  gc_DbmTranslation_de_Texts : ARRAY[0..2371] OF POINTER TO WSTRING(123) := [ADR(gc_DbmTranslation_de_Text0), ADR(gc_DbmTranslation_de_Text1), ADR(gc_DbmTranslation_de_Text2), ADR(gc_DbmTranslation_de_Text3), ADR(gc_DbmTranslation_de_Text4), ADR(gc_DbmTranslation_de_Text5), ADR(gc_DbmTranslation_de_Text6), ADR(gc_DbmTranslation_de_Text7), ADR(gc_DbmTranslation_de_Text8), ADR(gc_DbmTranslation_de_Text9), ADR(gc_DbmTranslation_de_Text10), ADR(gc_DbmTranslation_de_Text11), ADR(gc_DbmTranslation_de_Text12), ADR(gc_DbmTranslation_de_Text13), ADR(gc_DbmTranslation_de_Text14), ADR(gc_DbmTranslation_de_Text15), ADR(gc_DbmTranslation_de_Text16), ADR(gc_DbmTranslation_de_Text17), ADR(gc_DbmTranslation_de_Text18), ADR(gc_DbmTranslation_de_Text19), ADR(gc_DbmTranslation_de_Text20), ADR(gc_DbmTranslation_de_Text21), ADR(gc_DbmTranslation_de_Text22), ADR(gc_DbmTranslation_de_Text23), ADR(gc_DbmTranslation_de_Text24), ADR(gc_DbmTranslation_de_Text25), ADR(gc_DbmTranslation_de_Text26), ADR(gc_DbmTranslation_de_Text27), ADR(gc_DbmTranslation_de_Text28), ADR(gc_DbmTranslation_de_Text29), ADR(gc_DbmTranslation_de_Text30), ADR(gc_DbmTranslation_de_Text31), ADR(gc_DbmTranslation_de_Text32), ADR(gc_DbmTranslation_de_Text33), ADR(gc_DbmTranslation_de_Text34), ADR(gc_DbmTranslation_de_Text35), ADR(gc_DbmTranslation_de_Text36), ADR(gc_DbmTranslation_de_Text37), ADR(gc_DbmTranslation_de_Text38), ADR(gc_DbmTranslation_de_Text39), ADR(gc_DbmTranslation_de_Text40), ADR(gc_DbmTranslation_de_Text41), ADR(gc_DbmTranslation_de_Text42), ADR(gc_DbmTranslation_de_Text43), ADR(gc_DbmTranslation_de_Text44), ADR(gc_DbmTranslation_de_Text45), ADR(gc_DbmTranslation_de_Text46), ADR(gc_DbmTranslation_de_Text47), ADR(gc_DbmTranslation_de_Text48), ADR(gc_DbmTranslation_de_Text49), ADR(gc_DbmTranslation_de_Text50), ADR(gc_DbmTranslation_de_Text51), ADR(gc_DbmTranslation_de_Text52), ADR(gc_DbmTranslation_de_Text53), ADR(gc_DbmTranslation_de_Text54), ADR(gc_DbmTranslation_de_Text55), ADR(gc_DbmTranslation_de_Text56), ADR(gc_DbmTranslation_de_Text57), ADR(gc_DbmTranslation_de_Text58), ADR(gc_DbmTranslation_de_Text59), ADR(gc_DbmTranslation_de_Text60), ADR(gc_DbmTranslation_de_Text61), ADR(gc_DbmTranslation_de_Text62), ADR(gc_DbmTranslation_de_Text63), ADR(gc_DbmTranslation_de_Text64), ADR(gc_DbmTranslation_de_Text65), ADR(gc_DbmTranslation_de_Text66), ADR(gc_DbmTranslation_de_Text67), ADR(gc_DbmTranslation_de_Text68), ADR(gc_DbmTranslation_de_Text69), ADR(gc_DbmTranslation_de_Text70), ADR(gc_DbmTranslation_de_Text71), ADR(gc_DbmTranslation_de_Text72), ADR(gc_DbmTranslation_de_Text73), ADR(gc_DbmTranslation_de_Text74), ADR(gc_DbmTranslation_de_Text75), ADR(gc_DbmTranslation_de_Text76), ADR(gc_DbmTranslation_de_Text77), ADR(gc_DbmTranslation_de_Text78), ADR(gc_DbmTranslation_de_Text79), ADR(gc_DbmTranslation_de_Text80), ADR(gc_DbmTranslation_de_Text81), ADR(gc_DbmTranslation_de_Text82), ADR(gc_DbmTranslation_de_Text83), ADR(gc_DbmTranslation_de_Text84), ADR(gc_DbmTranslation_de_Text85), ADR(gc_DbmTranslation_de_Text86), ADR(gc_DbmTranslation_de_Text87), ADR(gc_DbmTranslation_de_Text88), ADR(gc_DbmTranslation_de_Text89), ADR(gc_DbmTranslation_de_Text90), ADR(gc_DbmTranslation_de_Text91), ADR(gc_DbmTranslation_de_Text92), ADR(gc_DbmTranslation_de_Text93), ADR(gc_DbmTranslation_de_Text94), ADR(gc_DbmTranslation_de_Text95), ADR(gc_DbmTranslation_de_Text96), ADR(gc_DbmTranslation_de_Text97), ADR(gc_DbmTranslation_de_Text98), ADR(gc_DbmTranslation_de_Text99), ADR(gc_DbmTranslation_de_Text100), ADR(gc_DbmTranslation_de_Text101), ADR(gc_DbmTranslation_de_Text102), ADR(gc_DbmTranslation_de_Text103), ADR(gc_DbmTranslation_de_Text104), ADR(gc_DbmTranslation_de_Text105), ADR(gc_DbmTranslation_de_Text106), ADR(gc_DbmTranslation_de_Text107), ADR(gc_DbmTranslation_de_Text108), ADR(gc_DbmTranslation_de_Text109), ADR(gc_DbmTranslation_de_Text110), ADR(gc_DbmTranslation_de_Text111), ADR(gc_DbmTranslation_de_Text112), ADR(gc_DbmTranslation_de_Text113), ADR(gc_DbmTranslation_de_Text114), ADR(gc_DbmTranslation_de_Text115), ADR(gc_DbmTranslation_de_Text116), ADR(gc_DbmTranslation_de_Text117), ADR(gc_DbmTranslation_de_Text118), ADR(gc_DbmTranslation_de_Text119), ADR(gc_DbmTranslation_de_Text120), ADR(gc_DbmTranslation_de_Text121), ADR(gc_DbmTranslation_de_Text122), ADR(gc_DbmTranslation_de_Text123), ADR(gc_DbmTranslation_de_Text124), ADR(gc_DbmTranslation_de_Text125), ADR(gc_DbmTranslation_de_Text126), ADR(gc_DbmTranslation_de_Text127), ADR(gc_DbmTranslation_de_Text128), ADR(gc_DbmTranslation_de_Text129), ADR(gc_DbmTranslation_de_Text130), ADR(gc_DbmTranslation_de_Text131), ADR(gc_DbmTranslation_de_Text132), ADR(gc_DbmTranslation_de_Text133), ADR(gc_DbmTranslation_de_Text134), ADR(gc_DbmTranslation_de_Text135), ADR(gc_DbmTranslation_de_Text136), ADR(gc_DbmTranslation_de_Text137), ADR(gc_DbmTranslation_de_Text138), ADR(gc_DbmTranslation_de_Text139), ADR(gc_DbmTranslation_de_Text140), ADR(gc_DbmTranslation_de_Text141), ADR(gc_DbmTranslation_de_Text142), ADR(gc_DbmTranslation_de_Text143), ADR(gc_DbmTranslation_de_Text144), ADR(gc_DbmTranslation_de_Text145), ADR(gc_DbmTranslation_de_Text146), ADR(gc_DbmTranslation_de_Text147), ADR(gc_DbmTranslation_de_Text148), ADR(gc_DbmTranslation_de_Text149), ADR(gc_DbmTranslation_de_Text150), ADR(gc_DbmTranslation_de_Text151), ADR(gc_DbmTranslation_de_Text152), ADR(gc_DbmTranslation_de_Text153), ADR(gc_DbmTranslation_de_Text154), ADR(gc_DbmTranslation_de_Text155), ADR(gc_DbmTranslation_de_Text156), ADR(gc_DbmTranslation_de_Text157), ADR(gc_DbmTranslation_de_Text158), ADR(gc_DbmTranslation_de_Text159), ADR(gc_DbmTranslation_de_Text160), ADR(gc_DbmTranslation_de_Text161), ADR(gc_DbmTranslation_de_Text162), ADR(gc_DbmTranslation_de_Text163), ADR(gc_DbmTranslation_de_Text164), ADR(gc_DbmTranslation_de_Text165), ADR(gc_DbmTranslation_de_Text166), ADR(gc_DbmTranslation_de_Text167), ADR(gc_DbmTranslation_de_Text168), ADR(gc_DbmTranslation_de_Text169), ADR(gc_DbmTranslation_de_Text170), ADR(gc_DbmTranslation_de_Text171), ADR(gc_DbmTranslation_de_Text172), ADR(gc_DbmTranslation_de_Text173), ADR(gc_DbmTranslation_de_Text174), ADR(gc_DbmTranslation_de_Text175), ADR(gc_DbmTranslation_de_Text176), ADR(gc_DbmTranslation_de_Text177), ADR(gc_DbmTranslation_de_Text178), ADR(gc_DbmTranslation_de_Text179), ADR(gc_DbmTranslation_de_Text180), ADR(gc_DbmTranslation_de_Text181), ADR(gc_DbmTranslation_de_Text182), ADR(gc_DbmTranslation_de_Text183), ADR(gc_DbmTranslation_de_Text184), ADR(gc_DbmTranslation_de_Text185), ADR(gc_DbmTranslation_de_Text186), ADR(gc_DbmTranslation_de_Text187), ADR(gc_DbmTranslation_de_Text188), ADR(gc_DbmTranslation_de_Text189), ADR(gc_DbmTranslation_de_Text190), ADR(gc_DbmTranslation_de_Text191), ADR(gc_DbmTranslation_de_Text192), ADR(gc_DbmTranslation_de_Text193), ADR(gc_DbmTranslation_de_Text194), ADR(gc_DbmTranslation_de_Text195), ADR(gc_DbmTranslation_de_Text196), ADR(gc_DbmTranslation_de_Text197), ADR(gc_DbmTranslation_de_Text198), ADR(gc_DbmTranslation_de_Text199), ADR(gc_DbmTranslation_de_Text200), ADR(gc_DbmTranslation_de_Text201), ADR(gc_DbmTranslation_de_Text202), ADR(gc_DbmTranslation_de_Text203), ADR(gc_DbmTranslation_de_Text204), ADR(gc_DbmTranslation_de_Text205), ADR(gc_DbmTranslation_de_Text206), ADR(gc_DbmTranslation_de_Text207), ADR(gc_DbmTranslation_de_Text208), ADR(gc_DbmTranslation_de_Text209), ADR(gc_DbmTranslation_de_Text210), ADR(gc_DbmTranslation_de_Text211), ADR(gc_DbmTranslation_de_Text212), ADR(gc_DbmTranslation_de_Text213), ADR(gc_DbmTranslation_de_Text214), ADR(gc_DbmTranslation_de_Text215), ADR(gc_DbmTranslation_de_Text216), ADR(gc_DbmTranslation_de_Text217), ADR(gc_DbmTranslation_de_Text218), ADR(gc_DbmTranslation_de_Text219), ADR(gc_DbmTranslation_de_Text220), ADR(gc_DbmTranslation_de_Text221), ADR(gc_DbmTranslation_de_Text222), ADR(gc_DbmTranslation_de_Text223), ADR(gc_DbmTranslation_de_Text224), ADR(gc_DbmTranslation_de_Text225), ADR(gc_DbmTranslation_de_Text226), ADR(gc_DbmTranslation_de_Text227), ADR(gc_DbmTranslation_de_Text228), ADR(gc_DbmTranslation_de_Text229), ADR(gc_DbmTranslation_de_Text230), ADR(gc_DbmTranslation_de_Text231), ADR(gc_DbmTranslation_de_Text232), ADR(gc_DbmTranslation_de_Text233), ADR(gc_DbmTranslation_de_Text234), ADR(gc_DbmTranslation_de_Text235), ADR(gc_DbmTranslation_de_Text236), ADR(gc_DbmTranslation_de_Text237), ADR(gc_DbmTranslation_de_Text238), ADR(gc_DbmTranslation_de_Text239), ADR(gc_DbmTranslation_de_Text240), ADR(gc_DbmTranslation_de_Text241), ADR(gc_DbmTranslation_de_Text242), ADR(gc_DbmTranslation_de_Text243), ADR(gc_DbmTranslation_de_Text244), ADR(gc_DbmTranslation_de_Text245), ADR(gc_DbmTranslation_de_Text246), ADR(gc_DbmTranslation_de_Text247), ADR(gc_DbmTranslation_de_Text248), ADR(gc_DbmTranslation_de_Text249), ADR(gc_DbmTranslation_de_Text250), ADR(gc_DbmTranslation_de_Text251), ADR(gc_DbmTranslation_de_Text252), ADR(gc_DbmTranslation_de_Text253), ADR(gc_DbmTranslation_de_Text254), ADR(gc_DbmTranslation_de_Text255), ADR(gc_DbmTranslation_de_Text256), ADR(gc_DbmTranslation_de_Text257), ADR(gc_DbmTranslation_de_Text258), ADR(gc_DbmTranslation_de_Text259), ADR(gc_DbmTranslation_de_Text260), ADR(gc_DbmTranslation_de_Text261), ADR(gc_DbmTranslation_de_Text262), ADR(gc_DbmTranslation_de_Text263), ADR(gc_DbmTranslation_de_Text264), ADR(gc_DbmTranslation_de_Text265), ADR(gc_DbmTranslation_de_Text266), ADR(gc_DbmTranslation_de_Text267), ADR(gc_DbmTranslation_de_Text268), ADR(gc_DbmTranslation_de_Text269), ADR(gc_DbmTranslation_de_Text270), ADR(gc_DbmTranslation_de_Text271), ADR(gc_DbmTranslation_de_Text272), ADR(gc_DbmTranslation_de_Text273), ADR(gc_DbmTranslation_de_Text274), ADR(gc_DbmTranslation_de_Text275), ADR(gc_DbmTranslation_de_Text276), ADR(gc_DbmTranslation_de_Text277), ADR(gc_DbmTranslation_de_Text278), ADR(gc_DbmTranslation_de_Text279), ADR(gc_DbmTranslation_de_Text280), ADR(gc_DbmTranslation_de_Text281), ADR(gc_DbmTranslation_de_Text282), ADR(gc_DbmTranslation_de_Text283), ADR(gc_DbmTranslation_de_Text284), ADR(gc_DbmTranslation_de_Text285), ADR(gc_DbmTranslation_de_Text286), ADR(gc_DbmTranslation_de_Text287), ADR(gc_DbmTranslation_de_Text288), ADR(gc_DbmTranslation_de_Text289), ADR(gc_DbmTranslation_de_Text290), ADR(gc_DbmTranslation_de_Text291), ADR(gc_DbmTranslation_de_Text292), ADR(gc_DbmTranslation_de_Text293), ADR(gc_DbmTranslation_de_Text294), ADR(gc_DbmTranslation_de_Text295), ADR(gc_DbmTranslation_de_Text296), ADR(gc_DbmTranslation_de_Text297), ADR(gc_DbmTranslation_de_Text298), ADR(gc_DbmTranslation_de_Text299), ADR(gc_DbmTranslation_de_Text300), ADR(gc_DbmTranslation_de_Text301), ADR(gc_DbmTranslation_de_Text302), ADR(gc_DbmTranslation_de_Text303), ADR(gc_DbmTranslation_de_Text304), ADR(gc_DbmTranslation_de_Text305), ADR(gc_DbmTranslation_de_Text306), ADR(gc_DbmTranslation_de_Text307), ADR(gc_DbmTranslation_de_Text308), ADR(gc_DbmTranslation_de_Text309), ADR(gc_DbmTranslation_de_Text310), ADR(gc_DbmTranslation_de_Text311), ADR(gc_DbmTranslation_de_Text312), ADR(gc_DbmTranslation_de_Text313), ADR(gc_DbmTranslation_de_Text314), ADR(gc_DbmTranslation_de_Text315), ADR(gc_DbmTranslation_de_Text316), ADR(gc_DbmTranslation_de_Text317), ADR(gc_DbmTranslation_de_Text318), ADR(gc_DbmTranslation_de_Text319), ADR(gc_DbmTranslation_de_Text320), ADR(gc_DbmTranslation_de_Text321), ADR(gc_DbmTranslation_de_Text322), ADR(gc_DbmTranslation_de_Text323), ADR(gc_DbmTranslation_de_Text324), ADR(gc_DbmTranslation_de_Text325), ADR(gc_DbmTranslation_de_Text326), ADR(gc_DbmTranslation_de_Text327), ADR(gc_DbmTranslation_de_Text328), ADR(gc_DbmTranslation_de_Text329), ADR(gc_DbmTranslation_de_Text330), ADR(gc_DbmTranslation_de_Text331), ADR(gc_DbmTranslation_de_Text332), ADR(gc_DbmTranslation_de_Text333), ADR(gc_DbmTranslation_de_Text334), ADR(gc_DbmTranslation_de_Text335), ADR(gc_DbmTranslation_de_Text336), ADR(gc_DbmTranslation_de_Text337), ADR(gc_DbmTranslation_de_Text338), ADR(gc_DbmTranslation_de_Text339), ADR(gc_DbmTranslation_de_Text340), ADR(gc_DbmTranslation_de_Text341), ADR(gc_DbmTranslation_de_Text342), ADR(gc_DbmTranslation_de_Text343), ADR(gc_DbmTranslation_de_Text344), ADR(gc_DbmTranslation_de_Text345), ADR(gc_DbmTranslation_de_Text346), ADR(gc_DbmTranslation_de_Text347), ADR(gc_DbmTranslation_de_Text348), ADR(gc_DbmTranslation_de_Text349), ADR(gc_DbmTranslation_de_Text350), ADR(gc_DbmTranslation_de_Text351), ADR(gc_DbmTranslation_de_Text352), ADR(gc_DbmTranslation_de_Text353), ADR(gc_DbmTranslation_de_Text354), ADR(gc_DbmTranslation_de_Text355), ADR(gc_DbmTranslation_de_Text356), ADR(gc_DbmTranslation_de_Text357), ADR(gc_DbmTranslation_de_Text358), ADR(gc_DbmTranslation_de_Text359), ADR(gc_DbmTranslation_de_Text360), ADR(gc_DbmTranslation_de_Text361), ADR(gc_DbmTranslation_de_Text362), ADR(gc_DbmTranslation_de_Text363), ADR(gc_DbmTranslation_de_Text364), ADR(gc_DbmTranslation_de_Text365), ADR(gc_DbmTranslation_de_Text366), ADR(gc_DbmTranslation_de_Text367), ADR(gc_DbmTranslation_de_Text368), ADR(gc_DbmTranslation_de_Text369), ADR(gc_DbmTranslation_de_Text370), ADR(gc_DbmTranslation_de_Text371), ADR(gc_DbmTranslation_de_Text372), ADR(gc_DbmTranslation_de_Text373), ADR(gc_DbmTranslation_de_Text374), ADR(gc_DbmTranslation_de_Text375), ADR(gc_DbmTranslation_de_Text376), ADR(gc_DbmTranslation_de_Text377), ADR(gc_DbmTranslation_de_Text378), ADR(gc_DbmTranslation_de_Text379), ADR(gc_DbmTranslation_de_Text380), ADR(gc_DbmTranslation_de_Text381), ADR(gc_DbmTranslation_de_Text382), ADR(gc_DbmTranslation_de_Text383), ADR(gc_DbmTranslation_de_Text384), ADR(gc_DbmTranslation_de_Text385), ADR(gc_DbmTranslation_de_Text386), ADR(gc_DbmTranslation_de_Text387), ADR(gc_DbmTranslation_de_Text388), ADR(gc_DbmTranslation_de_Text389), ADR(gc_DbmTranslation_de_Text390), ADR(gc_DbmTranslation_de_Text391), ADR(gc_DbmTranslation_de_Text392), ADR(gc_DbmTranslation_de_Text393), ADR(gc_DbmTranslation_de_Text394), ADR(gc_DbmTranslation_de_Text395), ADR(gc_DbmTranslation_de_Text396), ADR(gc_DbmTranslation_de_Text397), ADR(gc_DbmTranslation_de_Text398), ADR(gc_DbmTranslation_de_Text399), ADR(gc_DbmTranslation_de_Text400), ADR(gc_DbmTranslation_de_Text401), ADR(gc_DbmTranslation_de_Text402), ADR(gc_DbmTranslation_de_Text403), ADR(gc_DbmTranslation_de_Text404), ADR(gc_DbmTranslation_de_Text405), ADR(gc_DbmTranslation_de_Text406), ADR(gc_DbmTranslation_de_Text407), ADR(gc_DbmTranslation_de_Text408), ADR(gc_DbmTranslation_de_Text409), ADR(gc_DbmTranslation_de_Text410), ADR(gc_DbmTranslation_de_Text411), ADR(gc_DbmTranslation_de_Text412), ADR(gc_DbmTranslation_de_Text413), ADR(gc_DbmTranslation_de_Text414), ADR(gc_DbmTranslation_de_Text415), ADR(gc_DbmTranslation_de_Text416), ADR(gc_DbmTranslation_de_Text417), ADR(gc_DbmTranslation_de_Text418), ADR(gc_DbmTranslation_de_Text419), ADR(gc_DbmTranslation_de_Text420), ADR(gc_DbmTranslation_de_Text421), ADR(gc_DbmTranslation_de_Text422), ADR(gc_DbmTranslation_de_Text423), ADR(gc_DbmTranslation_de_Text424), ADR(gc_DbmTranslation_de_Text425), ADR(gc_DbmTranslation_de_Text426), ADR(gc_DbmTranslation_de_Text427), ADR(gc_DbmTranslation_de_Text428), ADR(gc_DbmTranslation_de_Text429), ADR(gc_DbmTranslation_de_Text430), ADR(gc_DbmTranslation_de_Text431), ADR(gc_DbmTranslation_de_Text432), ADR(gc_DbmTranslation_de_Text433), ADR(gc_DbmTranslation_de_Text434), ADR(gc_DbmTranslation_de_Text435), ADR(gc_DbmTranslation_de_Text436), ADR(gc_DbmTranslation_de_Text437), ADR(gc_DbmTranslation_de_Text438), ADR(gc_DbmTranslation_de_Text439), ADR(gc_DbmTranslation_de_Text440), ADR(gc_DbmTranslation_de_Text441), ADR(gc_DbmTranslation_de_Text442), ADR(gc_DbmTranslation_de_Text443), ADR(gc_DbmTranslation_de_Text444), ADR(gc_DbmTranslation_de_Text445), ADR(gc_DbmTranslation_de_Text446), ADR(gc_DbmTranslation_de_Text447), ADR(gc_DbmTranslation_de_Text448), ADR(gc_DbmTranslation_de_Text449), ADR(gc_DbmTranslation_de_Text450), ADR(gc_DbmTranslation_de_Text451), ADR(gc_DbmTranslation_de_Text452), ADR(gc_DbmTranslation_de_Text453), ADR(gc_DbmTranslation_de_Text454), ADR(gc_DbmTranslation_de_Text455), ADR(gc_DbmTranslation_de_Text456), ADR(gc_DbmTranslation_de_Text457), ADR(gc_DbmTranslation_de_Text458), ADR(gc_DbmTranslation_de_Text459), ADR(gc_DbmTranslation_de_Text460), ADR(gc_DbmTranslation_de_Text461), ADR(gc_DbmTranslation_de_Text462), ADR(gc_DbmTranslation_de_Text463), ADR(gc_DbmTranslation_de_Text464), ADR(gc_DbmTranslation_de_Text465), ADR(gc_DbmTranslation_de_Text466), ADR(gc_DbmTranslation_de_Text467), ADR(gc_DbmTranslation_de_Text468), ADR(gc_DbmTranslation_de_Text469), ADR(gc_DbmTranslation_de_Text470), ADR(gc_DbmTranslation_de_Text471), ADR(gc_DbmTranslation_de_Text472), ADR(gc_DbmTranslation_de_Text473), ADR(gc_DbmTranslation_de_Text474), ADR(gc_DbmTranslation_de_Text475), ADR(gc_DbmTranslation_de_Text476), ADR(gc_DbmTranslation_de_Text477), ADR(gc_DbmTranslation_de_Text478), ADR(gc_DbmTranslation_de_Text479), ADR(gc_DbmTranslation_de_Text480), ADR(gc_DbmTranslation_de_Text481), ADR(gc_DbmTranslation_de_Text482), ADR(gc_DbmTranslation_de_Text483), ADR(gc_DbmTranslation_de_Text484), ADR(gc_DbmTranslation_de_Text485), ADR(gc_DbmTranslation_de_Text486), ADR(gc_DbmTranslation_de_Text487), ADR(gc_DbmTranslation_de_Text488), ADR(gc_DbmTranslation_de_Text489), ADR(gc_DbmTranslation_de_Text490), ADR(gc_DbmTranslation_de_Text491), ADR(gc_DbmTranslation_de_Text492), ADR(gc_DbmTranslation_de_Text493), ADR(gc_DbmTranslation_de_Text494), ADR(gc_DbmTranslation_de_Text495), ADR(gc_DbmTranslation_de_Text496), ADR(gc_DbmTranslation_de_Text497), ADR(gc_DbmTranslation_de_Text498), ADR(gc_DbmTranslation_de_Text499), ADR(gc_DbmTranslation_de_Text500), ADR(gc_DbmTranslation_de_Text501), ADR(gc_DbmTranslation_de_Text502), ADR(gc_DbmTranslation_de_Text503), ADR(gc_DbmTranslation_de_Text504), ADR(gc_DbmTranslation_de_Text505), ADR(gc_DbmTranslation_de_Text506), ADR(gc_DbmTranslation_de_Text507), ADR(gc_DbmTranslation_de_Text508), ADR(gc_DbmTranslation_de_Text509), ADR(gc_DbmTranslation_de_Text510), ADR(gc_DbmTranslation_de_Text511), ADR(gc_DbmTranslation_de_Text512), ADR(gc_DbmTranslation_de_Text513), ADR(gc_DbmTranslation_de_Text514), ADR(gc_DbmTranslation_de_Text515), ADR(gc_DbmTranslation_de_Text516), ADR(gc_DbmTranslation_de_Text517), ADR(gc_DbmTranslation_de_Text518), ADR(gc_DbmTranslation_de_Text519), ADR(gc_DbmTranslation_de_Text520), ADR(gc_DbmTranslation_de_Text521), ADR(gc_DbmTranslation_de_Text522), ADR(gc_DbmTranslation_de_Text523), ADR(gc_DbmTranslation_de_Text524), ADR(gc_DbmTranslation_de_Text525), ADR(gc_DbmTranslation_de_Text526), ADR(gc_DbmTranslation_de_Text527), ADR(gc_DbmTranslation_de_Text528), ADR(gc_DbmTranslation_de_Text529), ADR(gc_DbmTranslation_de_Text530), ADR(gc_DbmTranslation_de_Text531), ADR(gc_DbmTranslation_de_Text532), ADR(gc_DbmTranslation_de_Text533), ADR(gc_DbmTranslation_de_Text534), ADR(gc_DbmTranslation_de_Text535), ADR(gc_DbmTranslation_de_Text536), ADR(gc_DbmTranslation_de_Text537), ADR(gc_DbmTranslation_de_Text538), ADR(gc_DbmTranslation_de_Text539), ADR(gc_DbmTranslation_de_Text540), ADR(gc_DbmTranslation_de_Text541), ADR(gc_DbmTranslation_de_Text542), ADR(gc_DbmTranslation_de_Text543), ADR(gc_DbmTranslation_de_Text544), ADR(gc_DbmTranslation_de_Text545), ADR(gc_DbmTranslation_de_Text546), ADR(gc_DbmTranslation_de_Text547), ADR(gc_DbmTranslation_de_Text548), ADR(gc_DbmTranslation_de_Text549), ADR(gc_DbmTranslation_de_Text550), ADR(gc_DbmTranslation_de_Text551), ADR(gc_DbmTranslation_de_Text552), ADR(gc_DbmTranslation_de_Text553), ADR(gc_DbmTranslation_de_Text554), ADR(gc_DbmTranslation_de_Text555), ADR(gc_DbmTranslation_de_Text556), ADR(gc_DbmTranslation_de_Text557), ADR(gc_DbmTranslation_de_Text558), ADR(gc_DbmTranslation_de_Text559), ADR(gc_DbmTranslation_de_Text560), ADR(gc_DbmTranslation_de_Text561), ADR(gc_DbmTranslation_de_Text562), ADR(gc_DbmTranslation_de_Text563), ADR(gc_DbmTranslation_de_Text564), ADR(gc_DbmTranslation_de_Text565), ADR(gc_DbmTranslation_de_Text566), ADR(gc_DbmTranslation_de_Text567), ADR(gc_DbmTranslation_de_Text568), ADR(gc_DbmTranslation_de_Text569), ADR(gc_DbmTranslation_de_Text570), ADR(gc_DbmTranslation_de_Text571), ADR(gc_DbmTranslation_de_Text572), ADR(gc_DbmTranslation_de_Text573), ADR(gc_DbmTranslation_de_Text574), ADR(gc_DbmTranslation_de_Text575), ADR(gc_DbmTranslation_de_Text576), ADR(gc_DbmTranslation_de_Text577), ADR(gc_DbmTranslation_de_Text578), ADR(gc_DbmTranslation_de_Text579), ADR(gc_DbmTranslation_de_Text580), ADR(gc_DbmTranslation_de_Text581), ADR(gc_DbmTranslation_de_Text582), ADR(gc_DbmTranslation_de_Text583), ADR(gc_DbmTranslation_de_Text584), ADR(gc_DbmTranslation_de_Text585), ADR(gc_DbmTranslation_de_Text586), ADR(gc_DbmTranslation_de_Text587), ADR(gc_DbmTranslation_de_Text588), ADR(gc_DbmTranslation_de_Text589), ADR(gc_DbmTranslation_de_Text590), ADR(gc_DbmTranslation_de_Text591), ADR(gc_DbmTranslation_de_Text592), ADR(gc_DbmTranslation_de_Text593), ADR(gc_DbmTranslation_de_Text594), ADR(gc_DbmTranslation_de_Text595), ADR(gc_DbmTranslation_de_Text596), ADR(gc_DbmTranslation_de_Text597), ADR(gc_DbmTranslation_de_Text598), ADR(gc_DbmTranslation_de_Text599), ADR(gc_DbmTranslation_de_Text600), ADR(gc_DbmTranslation_de_Text601), ADR(gc_DbmTranslation_de_Text602), ADR(gc_DbmTranslation_de_Text603), ADR(gc_DbmTranslation_de_Text604), ADR(gc_DbmTranslation_de_Text605), ADR(gc_DbmTranslation_de_Text606), ADR(gc_DbmTranslation_de_Text607), ADR(gc_DbmTranslation_de_Text608), ADR(gc_DbmTranslation_de_Text609), ADR(gc_DbmTranslation_de_Text610), ADR(gc_DbmTranslation_de_Text611), ADR(gc_DbmTranslation_de_Text612), ADR(gc_DbmTranslation_de_Text613), ADR(gc_DbmTranslation_de_Text614), ADR(gc_DbmTranslation_de_Text615), ADR(gc_DbmTranslation_de_Text616), ADR(gc_DbmTranslation_de_Text617), ADR(gc_DbmTranslation_de_Text618), ADR(gc_DbmTranslation_de_Text619), ADR(gc_DbmTranslation_de_Text620), ADR(gc_DbmTranslation_de_Text621), ADR(gc_DbmTranslation_de_Text622), ADR(gc_DbmTranslation_de_Text623), ADR(gc_DbmTranslation_de_Text624), ADR(gc_DbmTranslation_de_Text625), ADR(gc_DbmTranslation_de_Text626), ADR(gc_DbmTranslation_de_Text627), ADR(gc_DbmTranslation_de_Text628), ADR(gc_DbmTranslation_de_Text629), ADR(gc_DbmTranslation_de_Text630), ADR(gc_DbmTranslation_de_Text631), ADR(gc_DbmTranslation_de_Text632), ADR(gc_DbmTranslation_de_Text633), ADR(gc_DbmTranslation_de_Text634), ADR(gc_DbmTranslation_de_Text635), ADR(gc_DbmTranslation_de_Text636), ADR(gc_DbmTranslation_de_Text637), ADR(gc_DbmTranslation_de_Text638), ADR(gc_DbmTranslation_de_Text639), ADR(gc_DbmTranslation_de_Text640), ADR(gc_DbmTranslation_de_Text641), ADR(gc_DbmTranslation_de_Text642), ADR(gc_DbmTranslation_de_Text643), ADR(gc_DbmTranslation_de_Text644), ADR(gc_DbmTranslation_de_Text645), ADR(gc_DbmTranslation_de_Text646), ADR(gc_DbmTranslation_de_Text647), ADR(gc_DbmTranslation_de_Text648), ADR(gc_DbmTranslation_de_Text649), ADR(gc_DbmTranslation_de_Text650), ADR(gc_DbmTranslation_de_Text651), ADR(gc_DbmTranslation_de_Text652), ADR(gc_DbmTranslation_de_Text653), ADR(gc_DbmTranslation_de_Text654), ADR(gc_DbmTranslation_de_Text655), ADR(gc_DbmTranslation_de_Text656), ADR(gc_DbmTranslation_de_Text657), ADR(gc_DbmTranslation_de_Text658), ADR(gc_DbmTranslation_de_Text659), ADR(gc_DbmTranslation_de_Text660), ADR(gc_DbmTranslation_de_Text661), ADR(gc_DbmTranslation_de_Text662), ADR(gc_DbmTranslation_de_Text663), ADR(gc_DbmTranslation_de_Text664), ADR(gc_DbmTranslation_de_Text665), ADR(gc_DbmTranslation_de_Text666), ADR(gc_DbmTranslation_de_Text667), ADR(gc_DbmTranslation_de_Text668), ADR(gc_DbmTranslation_de_Text669), ADR(gc_DbmTranslation_de_Text670), ADR(gc_DbmTranslation_de_Text671), ADR(gc_DbmTranslation_de_Text672), ADR(gc_DbmTranslation_de_Text673), ADR(gc_DbmTranslation_de_Text674), ADR(gc_DbmTranslation_de_Text675), ADR(gc_DbmTranslation_de_Text676), ADR(gc_DbmTranslation_de_Text677), ADR(gc_DbmTranslation_de_Text678), ADR(gc_DbmTranslation_de_Text679), ADR(gc_DbmTranslation_de_Text680), ADR(gc_DbmTranslation_de_Text681), ADR(gc_DbmTranslation_de_Text682), ADR(gc_DbmTranslation_de_Text683), ADR(gc_DbmTranslation_de_Text684), ADR(gc_DbmTranslation_de_Text685), ADR(gc_DbmTranslation_de_Text686), ADR(gc_DbmTranslation_de_Text687), ADR(gc_DbmTranslation_de_Text688), ADR(gc_DbmTranslation_de_Text689), ADR(gc_DbmTranslation_de_Text690), ADR(gc_DbmTranslation_de_Text691), ADR(gc_DbmTranslation_de_Text692), ADR(gc_DbmTranslation_de_Text693), ADR(gc_DbmTranslation_de_Text694), ADR(gc_DbmTranslation_de_Text695), ADR(gc_DbmTranslation_de_Text696), ADR(gc_DbmTranslation_de_Text697), ADR(gc_DbmTranslation_de_Text698), ADR(gc_DbmTranslation_de_Text699), ADR(gc_DbmTranslation_de_Text700), ADR(gc_DbmTranslation_de_Text701), ADR(gc_DbmTranslation_de_Text702), ADR(gc_DbmTranslation_de_Text703), ADR(gc_DbmTranslation_de_Text704), ADR(gc_DbmTranslation_de_Text705), ADR(gc_DbmTranslation_de_Text706), ADR(gc_DbmTranslation_de_Text707), ADR(gc_DbmTranslation_de_Text708), ADR(gc_DbmTranslation_de_Text709), ADR(gc_DbmTranslation_de_Text710), ADR(gc_DbmTranslation_de_Text711), ADR(gc_DbmTranslation_de_Text712), ADR(gc_DbmTranslation_de_Text713), ADR(gc_DbmTranslation_de_Text714), ADR(gc_DbmTranslation_de_Text715), ADR(gc_DbmTranslation_de_Text716), ADR(gc_DbmTranslation_de_Text717), ADR(gc_DbmTranslation_de_Text718), ADR(gc_DbmTranslation_de_Text719), ADR(gc_DbmTranslation_de_Text720), ADR(gc_DbmTranslation_de_Text721), ADR(gc_DbmTranslation_de_Text722), ADR(gc_DbmTranslation_de_Text723), ADR(gc_DbmTranslation_de_Text724), ADR(gc_DbmTranslation_de_Text725), ADR(gc_DbmTranslation_de_Text726), ADR(gc_DbmTranslation_de_Text727), ADR(gc_DbmTranslation_de_Text728), ADR(gc_DbmTranslation_de_Text729), ADR(gc_DbmTranslation_de_Text730), ADR(gc_DbmTranslation_de_Text731), ADR(gc_DbmTranslation_de_Text732), ADR(gc_DbmTranslation_de_Text733), ADR(gc_DbmTranslation_de_Text734), ADR(gc_DbmTranslation_de_Text735), ADR(gc_DbmTranslation_de_Text736), ADR(gc_DbmTranslation_de_Text737), ADR(gc_DbmTranslation_de_Text738), ADR(gc_DbmTranslation_de_Text739), ADR(gc_DbmTranslation_de_Text740), ADR(gc_DbmTranslation_de_Text741), ADR(gc_DbmTranslation_de_Text742), ADR(gc_DbmTranslation_de_Text743), ADR(gc_DbmTranslation_de_Text744), ADR(gc_DbmTranslation_de_Text745), ADR(gc_DbmTranslation_de_Text746), ADR(gc_DbmTranslation_de_Text747), ADR(gc_DbmTranslation_de_Text748), ADR(gc_DbmTranslation_de_Text749), ADR(gc_DbmTranslation_de_Text750), ADR(gc_DbmTranslation_de_Text751), ADR(gc_DbmTranslation_de_Text752), ADR(gc_DbmTranslation_de_Text753), ADR(gc_DbmTranslation_de_Text754), ADR(gc_DbmTranslation_de_Text755), ADR(gc_DbmTranslation_de_Text756), ADR(gc_DbmTranslation_de_Text757), ADR(gc_DbmTranslation_de_Text758), ADR(gc_DbmTranslation_de_Text759), ADR(gc_DbmTranslation_de_Text760), ADR(gc_DbmTranslation_de_Text761), ADR(gc_DbmTranslation_de_Text762), ADR(gc_DbmTranslation_de_Text763), ADR(gc_DbmTranslation_de_Text764), ADR(gc_DbmTranslation_de_Text765), ADR(gc_DbmTranslation_de_Text766), ADR(gc_DbmTranslation_de_Text767), ADR(gc_DbmTranslation_de_Text768), ADR(gc_DbmTranslation_de_Text769), ADR(gc_DbmTranslation_de_Text770), ADR(gc_DbmTranslation_de_Text771), ADR(gc_DbmTranslation_de_Text772), ADR(gc_DbmTranslation_de_Text773), ADR(gc_DbmTranslation_de_Text774), ADR(gc_DbmTranslation_de_Text775), ADR(gc_DbmTranslation_de_Text776), ADR(gc_DbmTranslation_de_Text777), ADR(gc_DbmTranslation_de_Text778), ADR(gc_DbmTranslation_de_Text779), ADR(gc_DbmTranslation_de_Text780), ADR(gc_DbmTranslation_de_Text781), ADR(gc_DbmTranslation_de_Text782), ADR(gc_DbmTranslation_de_Text783), ADR(gc_DbmTranslation_de_Text784), ADR(gc_DbmTranslation_de_Text785), ADR(gc_DbmTranslation_de_Text786), ADR(gc_DbmTranslation_de_Text787), ADR(gc_DbmTranslation_de_Text788), ADR(gc_DbmTranslation_de_Text789), ADR(gc_DbmTranslation_de_Text790), ADR(gc_DbmTranslation_de_Text791), ADR(gc_DbmTranslation_de_Text792), ADR(gc_DbmTranslation_de_Text793), ADR(gc_DbmTranslation_de_Text794), ADR(gc_DbmTranslation_de_Text795), ADR(gc_DbmTranslation_de_Text796), ADR(gc_DbmTranslation_de_Text797), ADR(gc_DbmTranslation_de_Text798), ADR(gc_DbmTranslation_de_Text799), ADR(gc_DbmTranslation_de_Text800), ADR(gc_DbmTranslation_de_Text801), ADR(gc_DbmTranslation_de_Text802), ADR(gc_DbmTranslation_de_Text803), ADR(gc_DbmTranslation_de_Text804), ADR(gc_DbmTranslation_de_Text805), ADR(gc_DbmTranslation_de_Text806), ADR(gc_DbmTranslation_de_Text807), ADR(gc_DbmTranslation_de_Text808), ADR(gc_DbmTranslation_de_Text809), ADR(gc_DbmTranslation_de_Text810), ADR(gc_DbmTranslation_de_Text811), ADR(gc_DbmTranslation_de_Text812), ADR(gc_DbmTranslation_de_Text813), ADR(gc_DbmTranslation_de_Text814), ADR(gc_DbmTranslation_de_Text815), ADR(gc_DbmTranslation_de_Text816), ADR(gc_DbmTranslation_de_Text817), ADR(gc_DbmTranslation_de_Text818), ADR(gc_DbmTranslation_de_Text819), ADR(gc_DbmTranslation_de_Text820), ADR(gc_DbmTranslation_de_Text821), ADR(gc_DbmTranslation_de_Text822), ADR(gc_DbmTranslation_de_Text823), ADR(gc_DbmTranslation_de_Text824), ADR(gc_DbmTranslation_de_Text825), ADR(gc_DbmTranslation_de_Text826), ADR(gc_DbmTranslation_de_Text827), ADR(gc_DbmTranslation_de_Text828), ADR(gc_DbmTranslation_de_Text829), ADR(gc_DbmTranslation_de_Text830), ADR(gc_DbmTranslation_de_Text831), ADR(gc_DbmTranslation_de_Text832), ADR(gc_DbmTranslation_de_Text833), ADR(gc_DbmTranslation_de_Text834), ADR(gc_DbmTranslation_de_Text835), ADR(gc_DbmTranslation_de_Text836), ADR(gc_DbmTranslation_de_Text837), ADR(gc_DbmTranslation_de_Text838), ADR(gc_DbmTranslation_de_Text839), ADR(gc_DbmTranslation_de_Text840), ADR(gc_DbmTranslation_de_Text841), ADR(gc_DbmTranslation_de_Text842), ADR(gc_DbmTranslation_de_Text843), ADR(gc_DbmTranslation_de_Text844), ADR(gc_DbmTranslation_de_Text845), ADR(gc_DbmTranslation_de_Text846), ADR(gc_DbmTranslation_de_Text847), ADR(gc_DbmTranslation_de_Text848), ADR(gc_DbmTranslation_de_Text849), ADR(gc_DbmTranslation_de_Text850), ADR(gc_DbmTranslation_de_Text851), ADR(gc_DbmTranslation_de_Text852), ADR(gc_DbmTranslation_de_Text853), ADR(gc_DbmTranslation_de_Text854), ADR(gc_DbmTranslation_de_Text855), ADR(gc_DbmTranslation_de_Text856), ADR(gc_DbmTranslation_de_Text857), ADR(gc_DbmTranslation_de_Text858), ADR(gc_DbmTranslation_de_Text859), ADR(gc_DbmTranslation_de_Text860), ADR(gc_DbmTranslation_de_Text861), ADR(gc_DbmTranslation_de_Text862), ADR(gc_DbmTranslation_de_Text863), ADR(gc_DbmTranslation_de_Text864), ADR(gc_DbmTranslation_de_Text865), ADR(gc_DbmTranslation_de_Text866), ADR(gc_DbmTranslation_de_Text867), ADR(gc_DbmTranslation_de_Text868), ADR(gc_DbmTranslation_de_Text869), ADR(gc_DbmTranslation_de_Text870), ADR(gc_DbmTranslation_de_Text871), ADR(gc_DbmTranslation_de_Text872), ADR(gc_DbmTranslation_de_Text873), ADR(gc_DbmTranslation_de_Text874), ADR(gc_DbmTranslation_de_Text875), ADR(gc_DbmTranslation_de_Text876), ADR(gc_DbmTranslation_de_Text877), ADR(gc_DbmTranslation_de_Text878), ADR(gc_DbmTranslation_de_Text879), ADR(gc_DbmTranslation_de_Text880), ADR(gc_DbmTranslation_de_Text881), ADR(gc_DbmTranslation_de_Text882), ADR(gc_DbmTranslation_de_Text883), ADR(gc_DbmTranslation_de_Text884), ADR(gc_DbmTranslation_de_Text885), ADR(gc_DbmTranslation_de_Text886), ADR(gc_DbmTranslation_de_Text887), ADR(gc_DbmTranslation_de_Text888), ADR(gc_DbmTranslation_de_Text889), ADR(gc_DbmTranslation_de_Text890), ADR(gc_DbmTranslation_de_Text891), ADR(gc_DbmTranslation_de_Text892), ADR(gc_DbmTranslation_de_Text893), ADR(gc_DbmTranslation_de_Text894), ADR(gc_DbmTranslation_de_Text895), ADR(gc_DbmTranslation_de_Text896), ADR(gc_DbmTranslation_de_Text897), ADR(gc_DbmTranslation_de_Text898), ADR(gc_DbmTranslation_de_Text899), ADR(gc_DbmTranslation_de_Text900), ADR(gc_DbmTranslation_de_Text901), ADR(gc_DbmTranslation_de_Text902), ADR(gc_DbmTranslation_de_Text903), ADR(gc_DbmTranslation_de_Text904), ADR(gc_DbmTranslation_de_Text905), ADR(gc_DbmTranslation_de_Text906), ADR(gc_DbmTranslation_de_Text907), ADR(gc_DbmTranslation_de_Text908), ADR(gc_DbmTranslation_de_Text909), ADR(gc_DbmTranslation_de_Text910), ADR(gc_DbmTranslation_de_Text911), ADR(gc_DbmTranslation_de_Text912), ADR(gc_DbmTranslation_de_Text913), ADR(gc_DbmTranslation_de_Text914), ADR(gc_DbmTranslation_de_Text915), ADR(gc_DbmTranslation_de_Text916), ADR(gc_DbmTranslation_de_Text917), ADR(gc_DbmTranslation_de_Text918), ADR(gc_DbmTranslation_de_Text919), ADR(gc_DbmTranslation_de_Text920), ADR(gc_DbmTranslation_de_Text921), ADR(gc_DbmTranslation_de_Text922), ADR(gc_DbmTranslation_de_Text923), ADR(gc_DbmTranslation_de_Text924), ADR(gc_DbmTranslation_de_Text925), ADR(gc_DbmTranslation_de_Text926), ADR(gc_DbmTranslation_de_Text927), ADR(gc_DbmTranslation_de_Text928), ADR(gc_DbmTranslation_de_Text929), ADR(gc_DbmTranslation_de_Text930), ADR(gc_DbmTranslation_de_Text931), ADR(gc_DbmTranslation_de_Text932), ADR(gc_DbmTranslation_de_Text933), ADR(gc_DbmTranslation_de_Text934), ADR(gc_DbmTranslation_de_Text935), ADR(gc_DbmTranslation_de_Text936), ADR(gc_DbmTranslation_de_Text937), ADR(gc_DbmTranslation_de_Text938), ADR(gc_DbmTranslation_de_Text939), ADR(gc_DbmTranslation_de_Text940), ADR(gc_DbmTranslation_de_Text941), ADR(gc_DbmTranslation_de_Text942), ADR(gc_DbmTranslation_de_Text943), ADR(gc_DbmTranslation_de_Text944), ADR(gc_DbmTranslation_de_Text945), ADR(gc_DbmTranslation_de_Text946), ADR(gc_DbmTranslation_de_Text947), ADR(gc_DbmTranslation_de_Text948), ADR(gc_DbmTranslation_de_Text949), ADR(gc_DbmTranslation_de_Text950), ADR(gc_DbmTranslation_de_Text951), ADR(gc_DbmTranslation_de_Text952), ADR(gc_DbmTranslation_de_Text953), ADR(gc_DbmTranslation_de_Text954), ADR(gc_DbmTranslation_de_Text955), ADR(gc_DbmTranslation_de_Text956), ADR(gc_DbmTranslation_de_Text957), ADR(gc_DbmTranslation_de_Text958), ADR(gc_DbmTranslation_de_Text959), ADR(gc_DbmTranslation_de_Text960), ADR(gc_DbmTranslation_de_Text961), ADR(gc_DbmTranslation_de_Text962), ADR(gc_DbmTranslation_de_Text963), ADR(gc_DbmTranslation_de_Text964), ADR(gc_DbmTranslation_de_Text965), ADR(gc_DbmTranslation_de_Text966), ADR(gc_DbmTranslation_de_Text967), ADR(gc_DbmTranslation_de_Text968), ADR(gc_DbmTranslation_de_Text969), ADR(gc_DbmTranslation_de_Text970), ADR(gc_DbmTranslation_de_Text971), ADR(gc_DbmTranslation_de_Text972), ADR(gc_DbmTranslation_de_Text973), ADR(gc_DbmTranslation_de_Text974), ADR(gc_DbmTranslation_de_Text975), ADR(gc_DbmTranslation_de_Text976), ADR(gc_DbmTranslation_de_Text977), ADR(gc_DbmTranslation_de_Text978), ADR(gc_DbmTranslation_de_Text979), ADR(gc_DbmTranslation_de_Text980), ADR(gc_DbmTranslation_de_Text981), ADR(gc_DbmTranslation_de_Text982), ADR(gc_DbmTranslation_de_Text983), ADR(gc_DbmTranslation_de_Text984), ADR(gc_DbmTranslation_de_Text985), ADR(gc_DbmTranslation_de_Text986), ADR(gc_DbmTranslation_de_Text987), ADR(gc_DbmTranslation_de_Text988), ADR(gc_DbmTranslation_de_Text989), ADR(gc_DbmTranslation_de_Text990), ADR(gc_DbmTranslation_de_Text991), ADR(gc_DbmTranslation_de_Text992), ADR(gc_DbmTranslation_de_Text993), ADR(gc_DbmTranslation_de_Text994), ADR(gc_DbmTranslation_de_Text995), ADR(gc_DbmTranslation_de_Text996), ADR(gc_DbmTranslation_de_Text997), ADR(gc_DbmTranslation_de_Text998), ADR(gc_DbmTranslation_de_Text999), ADR(gc_DbmTranslation_de_Text1000), ADR(gc_DbmTranslation_de_Text1001), ADR(gc_DbmTranslation_de_Text1002), ADR(gc_DbmTranslation_de_Text1003), ADR(gc_DbmTranslation_de_Text1004), ADR(gc_DbmTranslation_de_Text1005), ADR(gc_DbmTranslation_de_Text1006), ADR(gc_DbmTranslation_de_Text1007), ADR(gc_DbmTranslation_de_Text1008), ADR(gc_DbmTranslation_de_Text1009), ADR(gc_DbmTranslation_de_Text1010), ADR(gc_DbmTranslation_de_Text1011), ADR(gc_DbmTranslation_de_Text1012), ADR(gc_DbmTranslation_de_Text1013), ADR(gc_DbmTranslation_de_Text1014), ADR(gc_DbmTranslation_de_Text1015), ADR(gc_DbmTranslation_de_Text1016), ADR(gc_DbmTranslation_de_Text1017), ADR(gc_DbmTranslation_de_Text1018), ADR(gc_DbmTranslation_de_Text1019), ADR(gc_DbmTranslation_de_Text1020), ADR(gc_DbmTranslation_de_Text1021), ADR(gc_DbmTranslation_de_Text1022), ADR(gc_DbmTranslation_de_Text1023), ADR(gc_DbmTranslation_de_Text1024), ADR(gc_DbmTranslation_de_Text1025), ADR(gc_DbmTranslation_de_Text1026), ADR(gc_DbmTranslation_de_Text1027), ADR(gc_DbmTranslation_de_Text1028), ADR(gc_DbmTranslation_de_Text1029), ADR(gc_DbmTranslation_de_Text1030), ADR(gc_DbmTranslation_de_Text1031), ADR(gc_DbmTranslation_de_Text1032), ADR(gc_DbmTranslation_de_Text1033), ADR(gc_DbmTranslation_de_Text1034), ADR(gc_DbmTranslation_de_Text1035), ADR(gc_DbmTranslation_de_Text1036), ADR(gc_DbmTranslation_de_Text1037), ADR(gc_DbmTranslation_de_Text1038), ADR(gc_DbmTranslation_de_Text1039), ADR(gc_DbmTranslation_de_Text1040), ADR(gc_DbmTranslation_de_Text1041), ADR(gc_DbmTranslation_de_Text1042), ADR(gc_DbmTranslation_de_Text1043), ADR(gc_DbmTranslation_de_Text1044), ADR(gc_DbmTranslation_de_Text1045), ADR(gc_DbmTranslation_de_Text1046), ADR(gc_DbmTranslation_de_Text1047), ADR(gc_DbmTranslation_de_Text1048), ADR(gc_DbmTranslation_de_Text1049), ADR(gc_DbmTranslation_de_Text1050), ADR(gc_DbmTranslation_de_Text1051), ADR(gc_DbmTranslation_de_Text1052), ADR(gc_DbmTranslation_de_Text1053), ADR(gc_DbmTranslation_de_Text1054), ADR(gc_DbmTranslation_de_Text1055), ADR(gc_DbmTranslation_de_Text1056), ADR(gc_DbmTranslation_de_Text1057), ADR(gc_DbmTranslation_de_Text1058), ADR(gc_DbmTranslation_de_Text1059), ADR(gc_DbmTranslation_de_Text1060), ADR(gc_DbmTranslation_de_Text1061), ADR(gc_DbmTranslation_de_Text1062), ADR(gc_DbmTranslation_de_Text1063), ADR(gc_DbmTranslation_de_Text1064), ADR(gc_DbmTranslation_de_Text1065), ADR(gc_DbmTranslation_de_Text1066), ADR(gc_DbmTranslation_de_Text1067), ADR(gc_DbmTranslation_de_Text1068), ADR(gc_DbmTranslation_de_Text1069), ADR(gc_DbmTranslation_de_Text1070), ADR(gc_DbmTranslation_de_Text1071), ADR(gc_DbmTranslation_de_Text1072), ADR(gc_DbmTranslation_de_Text1073), ADR(gc_DbmTranslation_de_Text1074), ADR(gc_DbmTranslation_de_Text1075), ADR(gc_DbmTranslation_de_Text1076), ADR(gc_DbmTranslation_de_Text1077), ADR(gc_DbmTranslation_de_Text1078), ADR(gc_DbmTranslation_de_Text1079), ADR(gc_DbmTranslation_de_Text1080), ADR(gc_DbmTranslation_de_Text1081), ADR(gc_DbmTranslation_de_Text1082), ADR(gc_DbmTranslation_de_Text1083), ADR(gc_DbmTranslation_de_Text1084), ADR(gc_DbmTranslation_de_Text1085), ADR(gc_DbmTranslation_de_Text1086), ADR(gc_DbmTranslation_de_Text1087), ADR(gc_DbmTranslation_de_Text1088), ADR(gc_DbmTranslation_de_Text1089), ADR(gc_DbmTranslation_de_Text1090), ADR(gc_DbmTranslation_de_Text1091), ADR(gc_DbmTranslation_de_Text1092), ADR(gc_DbmTranslation_de_Text1093), ADR(gc_DbmTranslation_de_Text1094), ADR(gc_DbmTranslation_de_Text1095), ADR(gc_DbmTranslation_de_Text1096), ADR(gc_DbmTranslation_de_Text1097), ADR(gc_DbmTranslation_de_Text1098), ADR(gc_DbmTranslation_de_Text1099), ADR(gc_DbmTranslation_de_Text1100), ADR(gc_DbmTranslation_de_Text1101), ADR(gc_DbmTranslation_de_Text1102), ADR(gc_DbmTranslation_de_Text1103), ADR(gc_DbmTranslation_de_Text1104), ADR(gc_DbmTranslation_de_Text1105), ADR(gc_DbmTranslation_de_Text1106), ADR(gc_DbmTranslation_de_Text1107), ADR(gc_DbmTranslation_de_Text1108), ADR(gc_DbmTranslation_de_Text1109), ADR(gc_DbmTranslation_de_Text1110), ADR(gc_DbmTranslation_de_Text1111), ADR(gc_DbmTranslation_de_Text1112), ADR(gc_DbmTranslation_de_Text1113), ADR(gc_DbmTranslation_de_Text1114), ADR(gc_DbmTranslation_de_Text1115), ADR(gc_DbmTranslation_de_Text1116), ADR(gc_DbmTranslation_de_Text1117), ADR(gc_DbmTranslation_de_Text1118), ADR(gc_DbmTranslation_de_Text1119), ADR(gc_DbmTranslation_de_Text1120), ADR(gc_DbmTranslation_de_Text1121), ADR(gc_DbmTranslation_de_Text1122), ADR(gc_DbmTranslation_de_Text1123), ADR(gc_DbmTranslation_de_Text1124), ADR(gc_DbmTranslation_de_Text1125), ADR(gc_DbmTranslation_de_Text1126), ADR(gc_DbmTranslation_de_Text1127), ADR(gc_DbmTranslation_de_Text1128), ADR(gc_DbmTranslation_de_Text1129), ADR(gc_DbmTranslation_de_Text1130), ADR(gc_DbmTranslation_de_Text1131), ADR(gc_DbmTranslation_de_Text1132), ADR(gc_DbmTranslation_de_Text1133), ADR(gc_DbmTranslation_de_Text1134), ADR(gc_DbmTranslation_de_Text1135), ADR(gc_DbmTranslation_de_Text1136), ADR(gc_DbmTranslation_de_Text1137), ADR(gc_DbmTranslation_de_Text1138), ADR(gc_DbmTranslation_de_Text1139), ADR(gc_DbmTranslation_de_Text1140), ADR(gc_DbmTranslation_de_Text1141), ADR(gc_DbmTranslation_de_Text1142), ADR(gc_DbmTranslation_de_Text1143), ADR(gc_DbmTranslation_de_Text1144), ADR(gc_DbmTranslation_de_Text1145), ADR(gc_DbmTranslation_de_Text1146), ADR(gc_DbmTranslation_de_Text1147), ADR(gc_DbmTranslation_de_Text1148), ADR(gc_DbmTranslation_de_Text1149), ADR(gc_DbmTranslation_de_Text1150), ADR(gc_DbmTranslation_de_Text1151), ADR(gc_DbmTranslation_de_Text1152), ADR(gc_DbmTranslation_de_Text1153), ADR(gc_DbmTranslation_de_Text1154), ADR(gc_DbmTranslation_de_Text1155), ADR(gc_DbmTranslation_de_Text1156), ADR(gc_DbmTranslation_de_Text1157), ADR(gc_DbmTranslation_de_Text1158), ADR(gc_DbmTranslation_de_Text1159), ADR(gc_DbmTranslation_de_Text1160), ADR(gc_DbmTranslation_de_Text1161), ADR(gc_DbmTranslation_de_Text1162), ADR(gc_DbmTranslation_de_Text1163), ADR(gc_DbmTranslation_de_Text1164), ADR(gc_DbmTranslation_de_Text1165), ADR(gc_DbmTranslation_de_Text1166), ADR(gc_DbmTranslation_de_Text1167), ADR(gc_DbmTranslation_de_Text1168), ADR(gc_DbmTranslation_de_Text1169), ADR(gc_DbmTranslation_de_Text1170), ADR(gc_DbmTranslation_de_Text1171), ADR(gc_DbmTranslation_de_Text1172), ADR(gc_DbmTranslation_de_Text1173), ADR(gc_DbmTranslation_de_Text1174), ADR(gc_DbmTranslation_de_Text1175), ADR(gc_DbmTranslation_de_Text1176), ADR(gc_DbmTranslation_de_Text1177), ADR(gc_DbmTranslation_de_Text1178), ADR(gc_DbmTranslation_de_Text1179), ADR(gc_DbmTranslation_de_Text1180), ADR(gc_DbmTranslation_de_Text1181), ADR(gc_DbmTranslation_de_Text1182), ADR(gc_DbmTranslation_de_Text1183), ADR(gc_DbmTranslation_de_Text1184), ADR(gc_DbmTranslation_de_Text1185), ADR(gc_DbmTranslation_de_Text1186), ADR(gc_DbmTranslation_de_Text1187), ADR(gc_DbmTranslation_de_Text1188), ADR(gc_DbmTranslation_de_Text1189), ADR(gc_DbmTranslation_de_Text1190), ADR(gc_DbmTranslation_de_Text1191), ADR(gc_DbmTranslation_de_Text1192), ADR(gc_DbmTranslation_de_Text1193), ADR(gc_DbmTranslation_de_Text1194), ADR(gc_DbmTranslation_de_Text1195), ADR(gc_DbmTranslation_de_Text1196), ADR(gc_DbmTranslation_de_Text1197), ADR(gc_DbmTranslation_de_Text1198), ADR(gc_DbmTranslation_de_Text1199), ADR(gc_DbmTranslation_de_Text1200), ADR(gc_DbmTranslation_de_Text1201), ADR(gc_DbmTranslation_de_Text1202), ADR(gc_DbmTranslation_de_Text1203), ADR(gc_DbmTranslation_de_Text1204), ADR(gc_DbmTranslation_de_Text1205), ADR(gc_DbmTranslation_de_Text1206), ADR(gc_DbmTranslation_de_Text1207), ADR(gc_DbmTranslation_de_Text1208), ADR(gc_DbmTranslation_de_Text1209), ADR(gc_DbmTranslation_de_Text1210), ADR(gc_DbmTranslation_de_Text1211), ADR(gc_DbmTranslation_de_Text1212), ADR(gc_DbmTranslation_de_Text1213), ADR(gc_DbmTranslation_de_Text1214), ADR(gc_DbmTranslation_de_Text1215), ADR(gc_DbmTranslation_de_Text1216), ADR(gc_DbmTranslation_de_Text1217), ADR(gc_DbmTranslation_de_Text1218), ADR(gc_DbmTranslation_de_Text1219), ADR(gc_DbmTranslation_de_Text1220), ADR(gc_DbmTranslation_de_Text1221), ADR(gc_DbmTranslation_de_Text1222), ADR(gc_DbmTranslation_de_Text1223), ADR(gc_DbmTranslation_de_Text1224), ADR(gc_DbmTranslation_de_Text1225), ADR(gc_DbmTranslation_de_Text1226), ADR(gc_DbmTranslation_de_Text1227), ADR(gc_DbmTranslation_de_Text1228), ADR(gc_DbmTranslation_de_Text1229), ADR(gc_DbmTranslation_de_Text1230), ADR(gc_DbmTranslation_de_Text1231), ADR(gc_DbmTranslation_de_Text1232), ADR(gc_DbmTranslation_de_Text1233), ADR(gc_DbmTranslation_de_Text1234), ADR(gc_DbmTranslation_de_Text1235), ADR(gc_DbmTranslation_de_Text1236), ADR(gc_DbmTranslation_de_Text1237), ADR(gc_DbmTranslation_de_Text1238), ADR(gc_DbmTranslation_de_Text1239), ADR(gc_DbmTranslation_de_Text1240), ADR(gc_DbmTranslation_de_Text1241), ADR(gc_DbmTranslation_de_Text1242), ADR(gc_DbmTranslation_de_Text1243), ADR(gc_DbmTranslation_de_Text1244), ADR(gc_DbmTranslation_de_Text1245), ADR(gc_DbmTranslation_de_Text1246), ADR(gc_DbmTranslation_de_Text1247), ADR(gc_DbmTranslation_de_Text1248), ADR(gc_DbmTranslation_de_Text1249), ADR(gc_DbmTranslation_de_Text1250), ADR(gc_DbmTranslation_de_Text1251), ADR(gc_DbmTranslation_de_Text1252), ADR(gc_DbmTranslation_de_Text1253), ADR(gc_DbmTranslation_de_Text1254), ADR(gc_DbmTranslation_de_Text1255), ADR(gc_DbmTranslation_de_Text1256), ADR(gc_DbmTranslation_de_Text1257), ADR(gc_DbmTranslation_de_Text1258), ADR(gc_DbmTranslation_de_Text1259), ADR(gc_DbmTranslation_de_Text1260), ADR(gc_DbmTranslation_de_Text1261), ADR(gc_DbmTranslation_de_Text1262), ADR(gc_DbmTranslation_de_Text1263), ADR(gc_DbmTranslation_de_Text1264), ADR(gc_DbmTranslation_de_Text1265), ADR(gc_DbmTranslation_de_Text1266), ADR(gc_DbmTranslation_de_Text1267), ADR(gc_DbmTranslation_de_Text1268), ADR(gc_DbmTranslation_de_Text1269), ADR(gc_DbmTranslation_de_Text1270), ADR(gc_DbmTranslation_de_Text1271), ADR(gc_DbmTranslation_de_Text1272), ADR(gc_DbmTranslation_de_Text1273), ADR(gc_DbmTranslation_de_Text1274), ADR(gc_DbmTranslation_de_Text1275), ADR(gc_DbmTranslation_de_Text1276), ADR(gc_DbmTranslation_de_Text1277), ADR(gc_DbmTranslation_de_Text1278), ADR(gc_DbmTranslation_de_Text1279), ADR(gc_DbmTranslation_de_Text1280), ADR(gc_DbmTranslation_de_Text1281), ADR(gc_DbmTranslation_de_Text1282), ADR(gc_DbmTranslation_de_Text1283), ADR(gc_DbmTranslation_de_Text1284), ADR(gc_DbmTranslation_de_Text1285), ADR(gc_DbmTranslation_de_Text1286), ADR(gc_DbmTranslation_de_Text1287), ADR(gc_DbmTranslation_de_Text1288), ADR(gc_DbmTranslation_de_Text1289), ADR(gc_DbmTranslation_de_Text1290), ADR(gc_DbmTranslation_de_Text1291), ADR(gc_DbmTranslation_de_Text1292), ADR(gc_DbmTranslation_de_Text1293), ADR(gc_DbmTranslation_de_Text1294), ADR(gc_DbmTranslation_de_Text1295), ADR(gc_DbmTranslation_de_Text1296), ADR(gc_DbmTranslation_de_Text1297), ADR(gc_DbmTranslation_de_Text1298), ADR(gc_DbmTranslation_de_Text1299), ADR(gc_DbmTranslation_de_Text1300), ADR(gc_DbmTranslation_de_Text1301), ADR(gc_DbmTranslation_de_Text1302), ADR(gc_DbmTranslation_de_Text1303), ADR(gc_DbmTranslation_de_Text1304), ADR(gc_DbmTranslation_de_Text1305), ADR(gc_DbmTranslation_de_Text1306), ADR(gc_DbmTranslation_de_Text1307), ADR(gc_DbmTranslation_de_Text1308), ADR(gc_DbmTranslation_de_Text1309), ADR(gc_DbmTranslation_de_Text1310), ADR(gc_DbmTranslation_de_Text1311), ADR(gc_DbmTranslation_de_Text1312), ADR(gc_DbmTranslation_de_Text1313), ADR(gc_DbmTranslation_de_Text1314), ADR(gc_DbmTranslation_de_Text1315), ADR(gc_DbmTranslation_de_Text1316), ADR(gc_DbmTranslation_de_Text1317), ADR(gc_DbmTranslation_de_Text1318), ADR(gc_DbmTranslation_de_Text1319), ADR(gc_DbmTranslation_de_Text1320), ADR(gc_DbmTranslation_de_Text1321), ADR(gc_DbmTranslation_de_Text1322), ADR(gc_DbmTranslation_de_Text1323), ADR(gc_DbmTranslation_de_Text1324), ADR(gc_DbmTranslation_de_Text1325), ADR(gc_DbmTranslation_de_Text1326), ADR(gc_DbmTranslation_de_Text1327), ADR(gc_DbmTranslation_de_Text1328), ADR(gc_DbmTranslation_de_Text1329), ADR(gc_DbmTranslation_de_Text1330), ADR(gc_DbmTranslation_de_Text1331), ADR(gc_DbmTranslation_de_Text1332), ADR(gc_DbmTranslation_de_Text1333), ADR(gc_DbmTranslation_de_Text1334), ADR(gc_DbmTranslation_de_Text1335), ADR(gc_DbmTranslation_de_Text1336), ADR(gc_DbmTranslation_de_Text1337), ADR(gc_DbmTranslation_de_Text1338), ADR(gc_DbmTranslation_de_Text1339), ADR(gc_DbmTranslation_de_Text1340), ADR(gc_DbmTranslation_de_Text1341), ADR(gc_DbmTranslation_de_Text1342), ADR(gc_DbmTranslation_de_Text1343), ADR(gc_DbmTranslation_de_Text1344), ADR(gc_DbmTranslation_de_Text1345), ADR(gc_DbmTranslation_de_Text1346), ADR(gc_DbmTranslation_de_Text1347), ADR(gc_DbmTranslation_de_Text1348), ADR(gc_DbmTranslation_de_Text1349), ADR(gc_DbmTranslation_de_Text1350), ADR(gc_DbmTranslation_de_Text1351), ADR(gc_DbmTranslation_de_Text1352), ADR(gc_DbmTranslation_de_Text1353), ADR(gc_DbmTranslation_de_Text1354), ADR(gc_DbmTranslation_de_Text1355), ADR(gc_DbmTranslation_de_Text1356), ADR(gc_DbmTranslation_de_Text1357), ADR(gc_DbmTranslation_de_Text1358), ADR(gc_DbmTranslation_de_Text1359), ADR(gc_DbmTranslation_de_Text1360), ADR(gc_DbmTranslation_de_Text1361), ADR(gc_DbmTranslation_de_Text1362), ADR(gc_DbmTranslation_de_Text1363), ADR(gc_DbmTranslation_de_Text1364), ADR(gc_DbmTranslation_de_Text1365), ADR(gc_DbmTranslation_de_Text1366), ADR(gc_DbmTranslation_de_Text1367), ADR(gc_DbmTranslation_de_Text1368), ADR(gc_DbmTranslation_de_Text1369), ADR(gc_DbmTranslation_de_Text1370), ADR(gc_DbmTranslation_de_Text1371), ADR(gc_DbmTranslation_de_Text1372), ADR(gc_DbmTranslation_de_Text1373), ADR(gc_DbmTranslation_de_Text1374), ADR(gc_DbmTranslation_de_Text1375), ADR(gc_DbmTranslation_de_Text1376), ADR(gc_DbmTranslation_de_Text1377), ADR(gc_DbmTranslation_de_Text1378), ADR(gc_DbmTranslation_de_Text1379), ADR(gc_DbmTranslation_de_Text1380), ADR(gc_DbmTranslation_de_Text1381), ADR(gc_DbmTranslation_de_Text1382), ADR(gc_DbmTranslation_de_Text1383), ADR(gc_DbmTranslation_de_Text1384), ADR(gc_DbmTranslation_de_Text1385), ADR(gc_DbmTranslation_de_Text1386), ADR(gc_DbmTranslation_de_Text1387), ADR(gc_DbmTranslation_de_Text1388), ADR(gc_DbmTranslation_de_Text1389), ADR(gc_DbmTranslation_de_Text1390), ADR(gc_DbmTranslation_de_Text1391), ADR(gc_DbmTranslation_de_Text1392), ADR(gc_DbmTranslation_de_Text1393), ADR(gc_DbmTranslation_de_Text1394), ADR(gc_DbmTranslation_de_Text1395), ADR(gc_DbmTranslation_de_Text1396), ADR(gc_DbmTranslation_de_Text1397), ADR(gc_DbmTranslation_de_Text1398), ADR(gc_DbmTranslation_de_Text1399), ADR(gc_DbmTranslation_de_Text1400), ADR(gc_DbmTranslation_de_Text1401), ADR(gc_DbmTranslation_de_Text1402), ADR(gc_DbmTranslation_de_Text1403), ADR(gc_DbmTranslation_de_Text1404), ADR(gc_DbmTranslation_de_Text1405), ADR(gc_DbmTranslation_de_Text1406), ADR(gc_DbmTranslation_de_Text1407), ADR(gc_DbmTranslation_de_Text1408), ADR(gc_DbmTranslation_de_Text1409), ADR(gc_DbmTranslation_de_Text1410), ADR(gc_DbmTranslation_de_Text1411), ADR(gc_DbmTranslation_de_Text1412), ADR(gc_DbmTranslation_de_Text1413), ADR(gc_DbmTranslation_de_Text1414), ADR(gc_DbmTranslation_de_Text1415), ADR(gc_DbmTranslation_de_Text1416), ADR(gc_DbmTranslation_de_Text1417), ADR(gc_DbmTranslation_de_Text1418), ADR(gc_DbmTranslation_de_Text1419), ADR(gc_DbmTranslation_de_Text1420), ADR(gc_DbmTranslation_de_Text1421), ADR(gc_DbmTranslation_de_Text1422), ADR(gc_DbmTranslation_de_Text1423), ADR(gc_DbmTranslation_de_Text1424), ADR(gc_DbmTranslation_de_Text1425), ADR(gc_DbmTranslation_de_Text1426), ADR(gc_DbmTranslation_de_Text1427), ADR(gc_DbmTranslation_de_Text1428), ADR(gc_DbmTranslation_de_Text1429), ADR(gc_DbmTranslation_de_Text1430), ADR(gc_DbmTranslation_de_Text1431), ADR(gc_DbmTranslation_de_Text1432), ADR(gc_DbmTranslation_de_Text1433), ADR(gc_DbmTranslation_de_Text1434), ADR(gc_DbmTranslation_de_Text1435), ADR(gc_DbmTranslation_de_Text1436), ADR(gc_DbmTranslation_de_Text1437), ADR(gc_DbmTranslation_de_Text1438), ADR(gc_DbmTranslation_de_Text1439), ADR(gc_DbmTranslation_de_Text1440), ADR(gc_DbmTranslation_de_Text1441), ADR(gc_DbmTranslation_de_Text1442), ADR(gc_DbmTranslation_de_Text1443), ADR(gc_DbmTranslation_de_Text1444), ADR(gc_DbmTranslation_de_Text1445), ADR(gc_DbmTranslation_de_Text1446), ADR(gc_DbmTranslation_de_Text1447), ADR(gc_DbmTranslation_de_Text1448), ADR(gc_DbmTranslation_de_Text1449), ADR(gc_DbmTranslation_de_Text1450), ADR(gc_DbmTranslation_de_Text1451), ADR(gc_DbmTranslation_de_Text1452), ADR(gc_DbmTranslation_de_Text1453), ADR(gc_DbmTranslation_de_Text1454), ADR(gc_DbmTranslation_de_Text1455), ADR(gc_DbmTranslation_de_Text1456), ADR(gc_DbmTranslation_de_Text1457), ADR(gc_DbmTranslation_de_Text1458), ADR(gc_DbmTranslation_de_Text1459), ADR(gc_DbmTranslation_de_Text1460), ADR(gc_DbmTranslation_de_Text1461), ADR(gc_DbmTranslation_de_Text1462), ADR(gc_DbmTranslation_de_Text1463), ADR(gc_DbmTranslation_de_Text1464), ADR(gc_DbmTranslation_de_Text1465), ADR(gc_DbmTranslation_de_Text1466), ADR(gc_DbmTranslation_de_Text1467), ADR(gc_DbmTranslation_de_Text1468), ADR(gc_DbmTranslation_de_Text1469), ADR(gc_DbmTranslation_de_Text1470), ADR(gc_DbmTranslation_de_Text1471), ADR(gc_DbmTranslation_de_Text1472), ADR(gc_DbmTranslation_de_Text1473), ADR(gc_DbmTranslation_de_Text1474), ADR(gc_DbmTranslation_de_Text1475), ADR(gc_DbmTranslation_de_Text1476), ADR(gc_DbmTranslation_de_Text1477), ADR(gc_DbmTranslation_de_Text1478), ADR(gc_DbmTranslation_de_Text1479), ADR(gc_DbmTranslation_de_Text1480), ADR(gc_DbmTranslation_de_Text1481), ADR(gc_DbmTranslation_de_Text1482), ADR(gc_DbmTranslation_de_Text1483), ADR(gc_DbmTranslation_de_Text1484), ADR(gc_DbmTranslation_de_Text1485), ADR(gc_DbmTranslation_de_Text1486), ADR(gc_DbmTranslation_de_Text1487), ADR(gc_DbmTranslation_de_Text1488), ADR(gc_DbmTranslation_de_Text1489), ADR(gc_DbmTranslation_de_Text1490), ADR(gc_DbmTranslation_de_Text1491), ADR(gc_DbmTranslation_de_Text1492), ADR(gc_DbmTranslation_de_Text1493), ADR(gc_DbmTranslation_de_Text1494), ADR(gc_DbmTranslation_de_Text1495), ADR(gc_DbmTranslation_de_Text1496), ADR(gc_DbmTranslation_de_Text1497), ADR(gc_DbmTranslation_de_Text1498), ADR(gc_DbmTranslation_de_Text1499), ADR(gc_DbmTranslation_de_Text1500), ADR(gc_DbmTranslation_de_Text1501), ADR(gc_DbmTranslation_de_Text1502), ADR(gc_DbmTranslation_de_Text1503), ADR(gc_DbmTranslation_de_Text1504), ADR(gc_DbmTranslation_de_Text1505), ADR(gc_DbmTranslation_de_Text1506), ADR(gc_DbmTranslation_de_Text1507), ADR(gc_DbmTranslation_de_Text1508), ADR(gc_DbmTranslation_de_Text1509), ADR(gc_DbmTranslation_de_Text1510), ADR(gc_DbmTranslation_de_Text1511), ADR(gc_DbmTranslation_de_Text1512), ADR(gc_DbmTranslation_de_Text1513), ADR(gc_DbmTranslation_de_Text1514), ADR(gc_DbmTranslation_de_Text1515), ADR(gc_DbmTranslation_de_Text1516), ADR(gc_DbmTranslation_de_Text1517), ADR(gc_DbmTranslation_de_Text1518), ADR(gc_DbmTranslation_de_Text1519), ADR(gc_DbmTranslation_de_Text1520), ADR(gc_DbmTranslation_de_Text1521), ADR(gc_DbmTranslation_de_Text1522), ADR(gc_DbmTranslation_de_Text1523), ADR(gc_DbmTranslation_de_Text1524), ADR(gc_DbmTranslation_de_Text1525), ADR(gc_DbmTranslation_de_Text1526), ADR(gc_DbmTranslation_de_Text1527), ADR(gc_DbmTranslation_de_Text1528), ADR(gc_DbmTranslation_de_Text1529), ADR(gc_DbmTranslation_de_Text1530), ADR(gc_DbmTranslation_de_Text1531), ADR(gc_DbmTranslation_de_Text1532), ADR(gc_DbmTranslation_de_Text1533), ADR(gc_DbmTranslation_de_Text1534), ADR(gc_DbmTranslation_de_Text1535), ADR(gc_DbmTranslation_de_Text1536), ADR(gc_DbmTranslation_de_Text1537), ADR(gc_DbmTranslation_de_Text1538), ADR(gc_DbmTranslation_de_Text1539), ADR(gc_DbmTranslation_de_Text1540), ADR(gc_DbmTranslation_de_Text1541), ADR(gc_DbmTranslation_de_Text1542), ADR(gc_DbmTranslation_de_Text1543), ADR(gc_DbmTranslation_de_Text1544), ADR(gc_DbmTranslation_de_Text1545), ADR(gc_DbmTranslation_de_Text1546), ADR(gc_DbmTranslation_de_Text1547), ADR(gc_DbmTranslation_de_Text1548), ADR(gc_DbmTranslation_de_Text1549), ADR(gc_DbmTranslation_de_Text1550), ADR(gc_DbmTranslation_de_Text1551), ADR(gc_DbmTranslation_de_Text1552), ADR(gc_DbmTranslation_de_Text1553), ADR(gc_DbmTranslation_de_Text1554), ADR(gc_DbmTranslation_de_Text1555), ADR(gc_DbmTranslation_de_Text1556), ADR(gc_DbmTranslation_de_Text1557), ADR(gc_DbmTranslation_de_Text1558), ADR(gc_DbmTranslation_de_Text1559), ADR(gc_DbmTranslation_de_Text1560), ADR(gc_DbmTranslation_de_Text1561), ADR(gc_DbmTranslation_de_Text1562), ADR(gc_DbmTranslation_de_Text1563), ADR(gc_DbmTranslation_de_Text1564), ADR(gc_DbmTranslation_de_Text1565), ADR(gc_DbmTranslation_de_Text1566), ADR(gc_DbmTranslation_de_Text1567), ADR(gc_DbmTranslation_de_Text1568), ADR(gc_DbmTranslation_de_Text1569), ADR(gc_DbmTranslation_de_Text1570), ADR(gc_DbmTranslation_de_Text1571), ADR(gc_DbmTranslation_de_Text1572), ADR(gc_DbmTranslation_de_Text1573), ADR(gc_DbmTranslation_de_Text1574), ADR(gc_DbmTranslation_de_Text1575), ADR(gc_DbmTranslation_de_Text1576), ADR(gc_DbmTranslation_de_Text1577), ADR(gc_DbmTranslation_de_Text1578), ADR(gc_DbmTranslation_de_Text1579), ADR(gc_DbmTranslation_de_Text1580), ADR(gc_DbmTranslation_de_Text1581), ADR(gc_DbmTranslation_de_Text1582), ADR(gc_DbmTranslation_de_Text1583), ADR(gc_DbmTranslation_de_Text1584), ADR(gc_DbmTranslation_de_Text1585), ADR(gc_DbmTranslation_de_Text1586), ADR(gc_DbmTranslation_de_Text1587), ADR(gc_DbmTranslation_de_Text1588), ADR(gc_DbmTranslation_de_Text1589), ADR(gc_DbmTranslation_de_Text1590), ADR(gc_DbmTranslation_de_Text1591), ADR(gc_DbmTranslation_de_Text1592), ADR(gc_DbmTranslation_de_Text1593), ADR(gc_DbmTranslation_de_Text1594), ADR(gc_DbmTranslation_de_Text1595), ADR(gc_DbmTranslation_de_Text1596), ADR(gc_DbmTranslation_de_Text1597), ADR(gc_DbmTranslation_de_Text1598), ADR(gc_DbmTranslation_de_Text1599), ADR(gc_DbmTranslation_de_Text1600), ADR(gc_DbmTranslation_de_Text1601), ADR(gc_DbmTranslation_de_Text1602), ADR(gc_DbmTranslation_de_Text1603), ADR(gc_DbmTranslation_de_Text1604), ADR(gc_DbmTranslation_de_Text1605), ADR(gc_DbmTranslation_de_Text1606), ADR(gc_DbmTranslation_de_Text1607), ADR(gc_DbmTranslation_de_Text1608), ADR(gc_DbmTranslation_de_Text1609), ADR(gc_DbmTranslation_de_Text1610), ADR(gc_DbmTranslation_de_Text1611), ADR(gc_DbmTranslation_de_Text1612), ADR(gc_DbmTranslation_de_Text1613), ADR(gc_DbmTranslation_de_Text1614), ADR(gc_DbmTranslation_de_Text1615), ADR(gc_DbmTranslation_de_Text1616), ADR(gc_DbmTranslation_de_Text1617), ADR(gc_DbmTranslation_de_Text1618), ADR(gc_DbmTranslation_de_Text1619), ADR(gc_DbmTranslation_de_Text1620), ADR(gc_DbmTranslation_de_Text1621), ADR(gc_DbmTranslation_de_Text1622), ADR(gc_DbmTranslation_de_Text1623), ADR(gc_DbmTranslation_de_Text1624), ADR(gc_DbmTranslation_de_Text1625), ADR(gc_DbmTranslation_de_Text1626), ADR(gc_DbmTranslation_de_Text1627), ADR(gc_DbmTranslation_de_Text1628), ADR(gc_DbmTranslation_de_Text1629), ADR(gc_DbmTranslation_de_Text1630), ADR(gc_DbmTranslation_de_Text1631), ADR(gc_DbmTranslation_de_Text1632), ADR(gc_DbmTranslation_de_Text1633), ADR(gc_DbmTranslation_de_Text1634), ADR(gc_DbmTranslation_de_Text1635), ADR(gc_DbmTranslation_de_Text1636), ADR(gc_DbmTranslation_de_Text1637), ADR(gc_DbmTranslation_de_Text1638), ADR(gc_DbmTranslation_de_Text1639), ADR(gc_DbmTranslation_de_Text1640), ADR(gc_DbmTranslation_de_Text1641), ADR(gc_DbmTranslation_de_Text1642), ADR(gc_DbmTranslation_de_Text1643), ADR(gc_DbmTranslation_de_Text1644), ADR(gc_DbmTranslation_de_Text1645), ADR(gc_DbmTranslation_de_Text1646), ADR(gc_DbmTranslation_de_Text1647), ADR(gc_DbmTranslation_de_Text1648), ADR(gc_DbmTranslation_de_Text1649), ADR(gc_DbmTranslation_de_Text1650), ADR(gc_DbmTranslation_de_Text1651), ADR(gc_DbmTranslation_de_Text1652), ADR(gc_DbmTranslation_de_Text1653), ADR(gc_DbmTranslation_de_Text1654), ADR(gc_DbmTranslation_de_Text1655), ADR(gc_DbmTranslation_de_Text1656), ADR(gc_DbmTranslation_de_Text1657), ADR(gc_DbmTranslation_de_Text1658), ADR(gc_DbmTranslation_de_Text1659), ADR(gc_DbmTranslation_de_Text1660), ADR(gc_DbmTranslation_de_Text1661), ADR(gc_DbmTranslation_de_Text1662), ADR(gc_DbmTranslation_de_Text1663), ADR(gc_DbmTranslation_de_Text1664), ADR(gc_DbmTranslation_de_Text1665), ADR(gc_DbmTranslation_de_Text1666), ADR(gc_DbmTranslation_de_Text1667), ADR(gc_DbmTranslation_de_Text1668), ADR(gc_DbmTranslation_de_Text1669), ADR(gc_DbmTranslation_de_Text1670), ADR(gc_DbmTranslation_de_Text1671), ADR(gc_DbmTranslation_de_Text1672), ADR(gc_DbmTranslation_de_Text1673), ADR(gc_DbmTranslation_de_Text1674), ADR(gc_DbmTranslation_de_Text1675), ADR(gc_DbmTranslation_de_Text1676), ADR(gc_DbmTranslation_de_Text1677), ADR(gc_DbmTranslation_de_Text1678), ADR(gc_DbmTranslation_de_Text1679), ADR(gc_DbmTranslation_de_Text1680), ADR(gc_DbmTranslation_de_Text1681), ADR(gc_DbmTranslation_de_Text1682), ADR(gc_DbmTranslation_de_Text1683), ADR(gc_DbmTranslation_de_Text1684), ADR(gc_DbmTranslation_de_Text1685), ADR(gc_DbmTranslation_de_Text1686), ADR(gc_DbmTranslation_de_Text1687), ADR(gc_DbmTranslation_de_Text1688), ADR(gc_DbmTranslation_de_Text1689), ADR(gc_DbmTranslation_de_Text1690), ADR(gc_DbmTranslation_de_Text1691), ADR(gc_DbmTranslation_de_Text1692), ADR(gc_DbmTranslation_de_Text1693), ADR(gc_DbmTranslation_de_Text1694), ADR(gc_DbmTranslation_de_Text1695), ADR(gc_DbmTranslation_de_Text1696), ADR(gc_DbmTranslation_de_Text1697), ADR(gc_DbmTranslation_de_Text1698), ADR(gc_DbmTranslation_de_Text1699), ADR(gc_DbmTranslation_de_Text1700), ADR(gc_DbmTranslation_de_Text1701), ADR(gc_DbmTranslation_de_Text1702), ADR(gc_DbmTranslation_de_Text1703), ADR(gc_DbmTranslation_de_Text1704), ADR(gc_DbmTranslation_de_Text1705), ADR(gc_DbmTranslation_de_Text1706), ADR(gc_DbmTranslation_de_Text1707), ADR(gc_DbmTranslation_de_Text1708), ADR(gc_DbmTranslation_de_Text1709), ADR(gc_DbmTranslation_de_Text1710), ADR(gc_DbmTranslation_de_Text1711), ADR(gc_DbmTranslation_de_Text1712), ADR(gc_DbmTranslation_de_Text1713), ADR(gc_DbmTranslation_de_Text1714), ADR(gc_DbmTranslation_de_Text1715), ADR(gc_DbmTranslation_de_Text1716), ADR(gc_DbmTranslation_de_Text1717), ADR(gc_DbmTranslation_de_Text1718), ADR(gc_DbmTranslation_de_Text1719), ADR(gc_DbmTranslation_de_Text1720), ADR(gc_DbmTranslation_de_Text1721), ADR(gc_DbmTranslation_de_Text1722), ADR(gc_DbmTranslation_de_Text1723), ADR(gc_DbmTranslation_de_Text1724), ADR(gc_DbmTranslation_de_Text1725), ADR(gc_DbmTranslation_de_Text1726), ADR(gc_DbmTranslation_de_Text1727), ADR(gc_DbmTranslation_de_Text1728), ADR(gc_DbmTranslation_de_Text1729), ADR(gc_DbmTranslation_de_Text1730), ADR(gc_DbmTranslation_de_Text1731), ADR(gc_DbmTranslation_de_Text1732), ADR(gc_DbmTranslation_de_Text1733), ADR(gc_DbmTranslation_de_Text1734), ADR(gc_DbmTranslation_de_Text1735), ADR(gc_DbmTranslation_de_Text1736), ADR(gc_DbmTranslation_de_Text1737), ADR(gc_DbmTranslation_de_Text1738), ADR(gc_DbmTranslation_de_Text1739), ADR(gc_DbmTranslation_de_Text1740), ADR(gc_DbmTranslation_de_Text1741), ADR(gc_DbmTranslation_de_Text1742), ADR(gc_DbmTranslation_de_Text1743), ADR(gc_DbmTranslation_de_Text1744), ADR(gc_DbmTranslation_de_Text1745), ADR(gc_DbmTranslation_de_Text1746), ADR(gc_DbmTranslation_de_Text1747), ADR(gc_DbmTranslation_de_Text1748), ADR(gc_DbmTranslation_de_Text1749), ADR(gc_DbmTranslation_de_Text1750), ADR(gc_DbmTranslation_de_Text1751), ADR(gc_DbmTranslation_de_Text1752), ADR(gc_DbmTranslation_de_Text1753), ADR(gc_DbmTranslation_de_Text1754), ADR(gc_DbmTranslation_de_Text1755), ADR(gc_DbmTranslation_de_Text1756), ADR(gc_DbmTranslation_de_Text1757), ADR(gc_DbmTranslation_de_Text1758), ADR(gc_DbmTranslation_de_Text1759), ADR(gc_DbmTranslation_de_Text1760), ADR(gc_DbmTranslation_de_Text1761), ADR(gc_DbmTranslation_de_Text1762), ADR(gc_DbmTranslation_de_Text1763), ADR(gc_DbmTranslation_de_Text1764), ADR(gc_DbmTranslation_de_Text1765), ADR(gc_DbmTranslation_de_Text1766), ADR(gc_DbmTranslation_de_Text1767), ADR(gc_DbmTranslation_de_Text1768), ADR(gc_DbmTranslation_de_Text1769), ADR(gc_DbmTranslation_de_Text1770), ADR(gc_DbmTranslation_de_Text1771), ADR(gc_DbmTranslation_de_Text1772), ADR(gc_DbmTranslation_de_Text1773), ADR(gc_DbmTranslation_de_Text1774), ADR(gc_DbmTranslation_de_Text1775), ADR(gc_DbmTranslation_de_Text1776), ADR(gc_DbmTranslation_de_Text1777), ADR(gc_DbmTranslation_de_Text1778), ADR(gc_DbmTranslation_de_Text1779), ADR(gc_DbmTranslation_de_Text1780), ADR(gc_DbmTranslation_de_Text1781), ADR(gc_DbmTranslation_de_Text1782), ADR(gc_DbmTranslation_de_Text1783), ADR(gc_DbmTranslation_de_Text1784), ADR(gc_DbmTranslation_de_Text1785), ADR(gc_DbmTranslation_de_Text1786), ADR(gc_DbmTranslation_de_Text1787), ADR(gc_DbmTranslation_de_Text1788), ADR(gc_DbmTranslation_de_Text1789), ADR(gc_DbmTranslation_de_Text1790), ADR(gc_DbmTranslation_de_Text1791), ADR(gc_DbmTranslation_de_Text1792), ADR(gc_DbmTranslation_de_Text1793), ADR(gc_DbmTranslation_de_Text1794), ADR(gc_DbmTranslation_de_Text1795), ADR(gc_DbmTranslation_de_Text1796), ADR(gc_DbmTranslation_de_Text1797), ADR(gc_DbmTranslation_de_Text1798), ADR(gc_DbmTranslation_de_Text1799), ADR(gc_DbmTranslation_de_Text1800), ADR(gc_DbmTranslation_de_Text1801), ADR(gc_DbmTranslation_de_Text1802), ADR(gc_DbmTranslation_de_Text1803), ADR(gc_DbmTranslation_de_Text1804), ADR(gc_DbmTranslation_de_Text1805), ADR(gc_DbmTranslation_de_Text1806), ADR(gc_DbmTranslation_de_Text1807), ADR(gc_DbmTranslation_de_Text1808), ADR(gc_DbmTranslation_de_Text1809), ADR(gc_DbmTranslation_de_Text1810), ADR(gc_DbmTranslation_de_Text1811), ADR(gc_DbmTranslation_de_Text1812), ADR(gc_DbmTranslation_de_Text1813), ADR(gc_DbmTranslation_de_Text1814), ADR(gc_DbmTranslation_de_Text1815), ADR(gc_DbmTranslation_de_Text1816), ADR(gc_DbmTranslation_de_Text1817), ADR(gc_DbmTranslation_de_Text1818), ADR(gc_DbmTranslation_de_Text1819), ADR(gc_DbmTranslation_de_Text1820), ADR(gc_DbmTranslation_de_Text1821), ADR(gc_DbmTranslation_de_Text1822), ADR(gc_DbmTranslation_de_Text1823), ADR(gc_DbmTranslation_de_Text1824), ADR(gc_DbmTranslation_de_Text1825), ADR(gc_DbmTranslation_de_Text1826), ADR(gc_DbmTranslation_de_Text1827), ADR(gc_DbmTranslation_de_Text1828), ADR(gc_DbmTranslation_de_Text1829), ADR(gc_DbmTranslation_de_Text1830), ADR(gc_DbmTranslation_de_Text1831), ADR(gc_DbmTranslation_de_Text1832), ADR(gc_DbmTranslation_de_Text1833), ADR(gc_DbmTranslation_de_Text1834), ADR(gc_DbmTranslation_de_Text1835), ADR(gc_DbmTranslation_de_Text1836), ADR(gc_DbmTranslation_de_Text1837), ADR(gc_DbmTranslation_de_Text1838), ADR(gc_DbmTranslation_de_Text1839), ADR(gc_DbmTranslation_de_Text1840), ADR(gc_DbmTranslation_de_Text1841), ADR(gc_DbmTranslation_de_Text1842), ADR(gc_DbmTranslation_de_Text1843), ADR(gc_DbmTranslation_de_Text1844), ADR(gc_DbmTranslation_de_Text1845), ADR(gc_DbmTranslation_de_Text1846), ADR(gc_DbmTranslation_de_Text1847), ADR(gc_DbmTranslation_de_Text1848), ADR(gc_DbmTranslation_de_Text1849), ADR(gc_DbmTranslation_de_Text1850), ADR(gc_DbmTranslation_de_Text1851), ADR(gc_DbmTranslation_de_Text1852), ADR(gc_DbmTranslation_de_Text1853), ADR(gc_DbmTranslation_de_Text1854), ADR(gc_DbmTranslation_de_Text1855), ADR(gc_DbmTranslation_de_Text1856), ADR(gc_DbmTranslation_de_Text1857), ADR(gc_DbmTranslation_de_Text1858), ADR(gc_DbmTranslation_de_Text1859), ADR(gc_DbmTranslation_de_Text1860), ADR(gc_DbmTranslation_de_Text1861), ADR(gc_DbmTranslation_de_Text1862), ADR(gc_DbmTranslation_de_Text1863), ADR(gc_DbmTranslation_de_Text1864), ADR(gc_DbmTranslation_de_Text1865), ADR(gc_DbmTranslation_de_Text1866), ADR(gc_DbmTranslation_de_Text1867), ADR(gc_DbmTranslation_de_Text1868), ADR(gc_DbmTranslation_de_Text1869), ADR(gc_DbmTranslation_de_Text1870), ADR(gc_DbmTranslation_de_Text1871), ADR(gc_DbmTranslation_de_Text1872), ADR(gc_DbmTranslation_de_Text1873), ADR(gc_DbmTranslation_de_Text1874), ADR(gc_DbmTranslation_de_Text1875), ADR(gc_DbmTranslation_de_Text1876), ADR(gc_DbmTranslation_de_Text1877), ADR(gc_DbmTranslation_de_Text1878), ADR(gc_DbmTranslation_de_Text1879), ADR(gc_DbmTranslation_de_Text1880), ADR(gc_DbmTranslation_de_Text1881), ADR(gc_DbmTranslation_de_Text1882), ADR(gc_DbmTranslation_de_Text1883), ADR(gc_DbmTranslation_de_Text1884), ADR(gc_DbmTranslation_de_Text1885), ADR(gc_DbmTranslation_de_Text1886), ADR(gc_DbmTranslation_de_Text1887), ADR(gc_DbmTranslation_de_Text1888), ADR(gc_DbmTranslation_de_Text1889), ADR(gc_DbmTranslation_de_Text1890), ADR(gc_DbmTranslation_de_Text1891), ADR(gc_DbmTranslation_de_Text1892), ADR(gc_DbmTranslation_de_Text1893), ADR(gc_DbmTranslation_de_Text1894), ADR(gc_DbmTranslation_de_Text1895), ADR(gc_DbmTranslation_de_Text1896), ADR(gc_DbmTranslation_de_Text1897), ADR(gc_DbmTranslation_de_Text1898), ADR(gc_DbmTranslation_de_Text1899), ADR(gc_DbmTranslation_de_Text1900), ADR(gc_DbmTranslation_de_Text1901), ADR(gc_DbmTranslation_de_Text1902), ADR(gc_DbmTranslation_de_Text1903), ADR(gc_DbmTranslation_de_Text1904), ADR(gc_DbmTranslation_de_Text1905), ADR(gc_DbmTranslation_de_Text1906), ADR(gc_DbmTranslation_de_Text1907), ADR(gc_DbmTranslation_de_Text1908), ADR(gc_DbmTranslation_de_Text1909), ADR(gc_DbmTranslation_de_Text1910), ADR(gc_DbmTranslation_de_Text1911), ADR(gc_DbmTranslation_de_Text1912), ADR(gc_DbmTranslation_de_Text1913), ADR(gc_DbmTranslation_de_Text1914), ADR(gc_DbmTranslation_de_Text1915), ADR(gc_DbmTranslation_de_Text1916), ADR(gc_DbmTranslation_de_Text1917), ADR(gc_DbmTranslation_de_Text1918), ADR(gc_DbmTranslation_de_Text1919), ADR(gc_DbmTranslation_de_Text1920), ADR(gc_DbmTranslation_de_Text1921), ADR(gc_DbmTranslation_de_Text1922), ADR(gc_DbmTranslation_de_Text1923), ADR(gc_DbmTranslation_de_Text1924), ADR(gc_DbmTranslation_de_Text1925), ADR(gc_DbmTranslation_de_Text1926), ADR(gc_DbmTranslation_de_Text1927), ADR(gc_DbmTranslation_de_Text1928), ADR(gc_DbmTranslation_de_Text1929), ADR(gc_DbmTranslation_de_Text1930), ADR(gc_DbmTranslation_de_Text1931), ADR(gc_DbmTranslation_de_Text1932), ADR(gc_DbmTranslation_de_Text1933), ADR(gc_DbmTranslation_de_Text1934), ADR(gc_DbmTranslation_de_Text1935), ADR(gc_DbmTranslation_de_Text1936), ADR(gc_DbmTranslation_de_Text1937), ADR(gc_DbmTranslation_de_Text1938), ADR(gc_DbmTranslation_de_Text1939), ADR(gc_DbmTranslation_de_Text1940), ADR(gc_DbmTranslation_de_Text1941), ADR(gc_DbmTranslation_de_Text1942), ADR(gc_DbmTranslation_de_Text1943), ADR(gc_DbmTranslation_de_Text1944), ADR(gc_DbmTranslation_de_Text1945), ADR(gc_DbmTranslation_de_Text1946), ADR(gc_DbmTranslation_de_Text1947), ADR(gc_DbmTranslation_de_Text1948), ADR(gc_DbmTranslation_de_Text1949), ADR(gc_DbmTranslation_de_Text1950), ADR(gc_DbmTranslation_de_Text1951), ADR(gc_DbmTranslation_de_Text1952), ADR(gc_DbmTranslation_de_Text1953), ADR(gc_DbmTranslation_de_Text1954), ADR(gc_DbmTranslation_de_Text1955), ADR(gc_DbmTranslation_de_Text1956), ADR(gc_DbmTranslation_de_Text1957), ADR(gc_DbmTranslation_de_Text1958), ADR(gc_DbmTranslation_de_Text1959), ADR(gc_DbmTranslation_de_Text1960), ADR(gc_DbmTranslation_de_Text1961), ADR(gc_DbmTranslation_de_Text1962), ADR(gc_DbmTranslation_de_Text1963), ADR(gc_DbmTranslation_de_Text1964), ADR(gc_DbmTranslation_de_Text1965), ADR(gc_DbmTranslation_de_Text1966), ADR(gc_DbmTranslation_de_Text1967), ADR(gc_DbmTranslation_de_Text1968), ADR(gc_DbmTranslation_de_Text1969), ADR(gc_DbmTranslation_de_Text1970), ADR(gc_DbmTranslation_de_Text1971), ADR(gc_DbmTranslation_de_Text1972), ADR(gc_DbmTranslation_de_Text1973), ADR(gc_DbmTranslation_de_Text1974), ADR(gc_DbmTranslation_de_Text1975), ADR(gc_DbmTranslation_de_Text1976), ADR(gc_DbmTranslation_de_Text1977), ADR(gc_DbmTranslation_de_Text1978), ADR(gc_DbmTranslation_de_Text1979), ADR(gc_DbmTranslation_de_Text1980), ADR(gc_DbmTranslation_de_Text1981), ADR(gc_DbmTranslation_de_Text1982), ADR(gc_DbmTranslation_de_Text1983), ADR(gc_DbmTranslation_de_Text1984), ADR(gc_DbmTranslation_de_Text1985), ADR(gc_DbmTranslation_de_Text1986), ADR(gc_DbmTranslation_de_Text1987), ADR(gc_DbmTranslation_de_Text1988), ADR(gc_DbmTranslation_de_Text1989), ADR(gc_DbmTranslation_de_Text1990), ADR(gc_DbmTranslation_de_Text1991), ADR(gc_DbmTranslation_de_Text1992), ADR(gc_DbmTranslation_de_Text1993), ADR(gc_DbmTranslation_de_Text1994), ADR(gc_DbmTranslation_de_Text1995), ADR(gc_DbmTranslation_de_Text1996), ADR(gc_DbmTranslation_de_Text1997), ADR(gc_DbmTranslation_de_Text1998), ADR(gc_DbmTranslation_de_Text1999), ADR(gc_DbmTranslation_de_Text2000), ADR(gc_DbmTranslation_de_Text2001), ADR(gc_DbmTranslation_de_Text2002), ADR(gc_DbmTranslation_de_Text2003), ADR(gc_DbmTranslation_de_Text2004), ADR(gc_DbmTranslation_de_Text2005), ADR(gc_DbmTranslation_de_Text2006), ADR(gc_DbmTranslation_de_Text2007), ADR(gc_DbmTranslation_de_Text2008), ADR(gc_DbmTranslation_de_Text2009), ADR(gc_DbmTranslation_de_Text2010), ADR(gc_DbmTranslation_de_Text2011), ADR(gc_DbmTranslation_de_Text2012), ADR(gc_DbmTranslation_de_Text2013), ADR(gc_DbmTranslation_de_Text2014), ADR(gc_DbmTranslation_de_Text2015), ADR(gc_DbmTranslation_de_Text2016), ADR(gc_DbmTranslation_de_Text2017), ADR(gc_DbmTranslation_de_Text2018), ADR(gc_DbmTranslation_de_Text2019), ADR(gc_DbmTranslation_de_Text2020), ADR(gc_DbmTranslation_de_Text2021), ADR(gc_DbmTranslation_de_Text2022), ADR(gc_DbmTranslation_de_Text2023), ADR(gc_DbmTranslation_de_Text2024), ADR(gc_DbmTranslation_de_Text2025), ADR(gc_DbmTranslation_de_Text2026), ADR(gc_DbmTranslation_de_Text2027), ADR(gc_DbmTranslation_de_Text2028), ADR(gc_DbmTranslation_de_Text2029), ADR(gc_DbmTranslation_de_Text2030), ADR(gc_DbmTranslation_de_Text2031), ADR(gc_DbmTranslation_de_Text2032), ADR(gc_DbmTranslation_de_Text2033), ADR(gc_DbmTranslation_de_Text2034), ADR(gc_DbmTranslation_de_Text2035), ADR(gc_DbmTranslation_de_Text2036), ADR(gc_DbmTranslation_de_Text2037), ADR(gc_DbmTranslation_de_Text2038), ADR(gc_DbmTranslation_de_Text2039), ADR(gc_DbmTranslation_de_Text2040), ADR(gc_DbmTranslation_de_Text2041), ADR(gc_DbmTranslation_de_Text2042), ADR(gc_DbmTranslation_de_Text2043), ADR(gc_DbmTranslation_de_Text2044), ADR(gc_DbmTranslation_de_Text2045), ADR(gc_DbmTranslation_de_Text2046), ADR(gc_DbmTranslation_de_Text2047), ADR(gc_DbmTranslation_de_Text2048), ADR(gc_DbmTranslation_de_Text2049), ADR(gc_DbmTranslation_de_Text2050), ADR(gc_DbmTranslation_de_Text2051), ADR(gc_DbmTranslation_de_Text2052), ADR(gc_DbmTranslation_de_Text2053), ADR(gc_DbmTranslation_de_Text2054), ADR(gc_DbmTranslation_de_Text2055), ADR(gc_DbmTranslation_de_Text2056), ADR(gc_DbmTranslation_de_Text2057), ADR(gc_DbmTranslation_de_Text2058), ADR(gc_DbmTranslation_de_Text2059), ADR(gc_DbmTranslation_de_Text2060), ADR(gc_DbmTranslation_de_Text2061), ADR(gc_DbmTranslation_de_Text2062), ADR(gc_DbmTranslation_de_Text2063), ADR(gc_DbmTranslation_de_Text2064), ADR(gc_DbmTranslation_de_Text2065), ADR(gc_DbmTranslation_de_Text2066), ADR(gc_DbmTranslation_de_Text2067), ADR(gc_DbmTranslation_de_Text2068), ADR(gc_DbmTranslation_de_Text2069), ADR(gc_DbmTranslation_de_Text2070), ADR(gc_DbmTranslation_de_Text2071), ADR(gc_DbmTranslation_de_Text2072), ADR(gc_DbmTranslation_de_Text2073), ADR(gc_DbmTranslation_de_Text2074), ADR(gc_DbmTranslation_de_Text2075), ADR(gc_DbmTranslation_de_Text2076), ADR(gc_DbmTranslation_de_Text2077), ADR(gc_DbmTranslation_de_Text2078), ADR(gc_DbmTranslation_de_Text2079), ADR(gc_DbmTranslation_de_Text2080), ADR(gc_DbmTranslation_de_Text2081), ADR(gc_DbmTranslation_de_Text2082), ADR(gc_DbmTranslation_de_Text2083), ADR(gc_DbmTranslation_de_Text2084), ADR(gc_DbmTranslation_de_Text2085), ADR(gc_DbmTranslation_de_Text2086), ADR(gc_DbmTranslation_de_Text2087), ADR(gc_DbmTranslation_de_Text2088), ADR(gc_DbmTranslation_de_Text2089), ADR(gc_DbmTranslation_de_Text2090), ADR(gc_DbmTranslation_de_Text2091), ADR(gc_DbmTranslation_de_Text2092), ADR(gc_DbmTranslation_de_Text2093), ADR(gc_DbmTranslation_de_Text2094), ADR(gc_DbmTranslation_de_Text2095), ADR(gc_DbmTranslation_de_Text2096), ADR(gc_DbmTranslation_de_Text2097), ADR(gc_DbmTranslation_de_Text2098), ADR(gc_DbmTranslation_de_Text2099), ADR(gc_DbmTranslation_de_Text2100), ADR(gc_DbmTranslation_de_Text2101), ADR(gc_DbmTranslation_de_Text2102), ADR(gc_DbmTranslation_de_Text2103), ADR(gc_DbmTranslation_de_Text2104), ADR(gc_DbmTranslation_de_Text2105), ADR(gc_DbmTranslation_de_Text2106), ADR(gc_DbmTranslation_de_Text2107), ADR(gc_DbmTranslation_de_Text2108), ADR(gc_DbmTranslation_de_Text2109), ADR(gc_DbmTranslation_de_Text2110), ADR(gc_DbmTranslation_de_Text2111), ADR(gc_DbmTranslation_de_Text2112), ADR(gc_DbmTranslation_de_Text2113), ADR(gc_DbmTranslation_de_Text2114), ADR(gc_DbmTranslation_de_Text2115), ADR(gc_DbmTranslation_de_Text2116), ADR(gc_DbmTranslation_de_Text2117), ADR(gc_DbmTranslation_de_Text2118), ADR(gc_DbmTranslation_de_Text2119), ADR(gc_DbmTranslation_de_Text2120), ADR(gc_DbmTranslation_de_Text2121), ADR(gc_DbmTranslation_de_Text2122), ADR(gc_DbmTranslation_de_Text2123), ADR(gc_DbmTranslation_de_Text2124), ADR(gc_DbmTranslation_de_Text2125), ADR(gc_DbmTranslation_de_Text2126), ADR(gc_DbmTranslation_de_Text2127), ADR(gc_DbmTranslation_de_Text2128), ADR(gc_DbmTranslation_de_Text2129), ADR(gc_DbmTranslation_de_Text2130), ADR(gc_DbmTranslation_de_Text2131), ADR(gc_DbmTranslation_de_Text2132), ADR(gc_DbmTranslation_de_Text2133), ADR(gc_DbmTranslation_de_Text2134), ADR(gc_DbmTranslation_de_Text2135), ADR(gc_DbmTranslation_de_Text2136), ADR(gc_DbmTranslation_de_Text2137), ADR(gc_DbmTranslation_de_Text2138), ADR(gc_DbmTranslation_de_Text2139), ADR(gc_DbmTranslation_de_Text2140), ADR(gc_DbmTranslation_de_Text2141), ADR(gc_DbmTranslation_de_Text2142), ADR(gc_DbmTranslation_de_Text2143), ADR(gc_DbmTranslation_de_Text2144), ADR(gc_DbmTranslation_de_Text2145), ADR(gc_DbmTranslation_de_Text2146), ADR(gc_DbmTranslation_de_Text2147), ADR(gc_DbmTranslation_de_Text2148), ADR(gc_DbmTranslation_de_Text2149), ADR(gc_DbmTranslation_de_Text2150), ADR(gc_DbmTranslation_de_Text2151), ADR(gc_DbmTranslation_de_Text2152), ADR(gc_DbmTranslation_de_Text2153), ADR(gc_DbmTranslation_de_Text2154), ADR(gc_DbmTranslation_de_Text2155), ADR(gc_DbmTranslation_de_Text2156), ADR(gc_DbmTranslation_de_Text2157), ADR(gc_DbmTranslation_de_Text2158), ADR(gc_DbmTranslation_de_Text2159), ADR(gc_DbmTranslation_de_Text2160), ADR(gc_DbmTranslation_de_Text2161), ADR(gc_DbmTranslation_de_Text2162), ADR(gc_DbmTranslation_de_Text2163), ADR(gc_DbmTranslation_de_Text2164), ADR(gc_DbmTranslation_de_Text2165), ADR(gc_DbmTranslation_de_Text2166), ADR(gc_DbmTranslation_de_Text2167), ADR(gc_DbmTranslation_de_Text2168), ADR(gc_DbmTranslation_de_Text2169), ADR(gc_DbmTranslation_de_Text2170), ADR(gc_DbmTranslation_de_Text2171), ADR(gc_DbmTranslation_de_Text2172), ADR(gc_DbmTranslation_de_Text2173), ADR(gc_DbmTranslation_de_Text2174), ADR(gc_DbmTranslation_de_Text2175), ADR(gc_DbmTranslation_de_Text2176), ADR(gc_DbmTranslation_de_Text2177), ADR(gc_DbmTranslation_de_Text2178), ADR(gc_DbmTranslation_de_Text2179), ADR(gc_DbmTranslation_de_Text2180), ADR(gc_DbmTranslation_de_Text2181), ADR(gc_DbmTranslation_de_Text2182), ADR(gc_DbmTranslation_de_Text2183), ADR(gc_DbmTranslation_de_Text2184), ADR(gc_DbmTranslation_de_Text2185), ADR(gc_DbmTranslation_de_Text2186), ADR(gc_DbmTranslation_de_Text2187), ADR(gc_DbmTranslation_de_Text2188), ADR(gc_DbmTranslation_de_Text2189), ADR(gc_DbmTranslation_de_Text2190), ADR(gc_DbmTranslation_de_Text2191), ADR(gc_DbmTranslation_de_Text2192), ADR(gc_DbmTranslation_de_Text2193), ADR(gc_DbmTranslation_de_Text2194), ADR(gc_DbmTranslation_de_Text2195), ADR(gc_DbmTranslation_de_Text2196), ADR(gc_DbmTranslation_de_Text2197), ADR(gc_DbmTranslation_de_Text2198), ADR(gc_DbmTranslation_de_Text2199), ADR(gc_DbmTranslation_de_Text2200), ADR(gc_DbmTranslation_de_Text2201), ADR(gc_DbmTranslation_de_Text2202), ADR(gc_DbmTranslation_de_Text2203), ADR(gc_DbmTranslation_de_Text2204), ADR(gc_DbmTranslation_de_Text2205), ADR(gc_DbmTranslation_de_Text2206), ADR(gc_DbmTranslation_de_Text2207), ADR(gc_DbmTranslation_de_Text2208), ADR(gc_DbmTranslation_de_Text2209), ADR(gc_DbmTranslation_de_Text2210), ADR(gc_DbmTranslation_de_Text2211), ADR(gc_DbmTranslation_de_Text2212), ADR(gc_DbmTranslation_de_Text2213), ADR(gc_DbmTranslation_de_Text2214), ADR(gc_DbmTranslation_de_Text2215), ADR(gc_DbmTranslation_de_Text2216), ADR(gc_DbmTranslation_de_Text2217), ADR(gc_DbmTranslation_de_Text2218), ADR(gc_DbmTranslation_de_Text2219), ADR(gc_DbmTranslation_de_Text2220), ADR(gc_DbmTranslation_de_Text2221), ADR(gc_DbmTranslation_de_Text2222), ADR(gc_DbmTranslation_de_Text2223), ADR(gc_DbmTranslation_de_Text2224), ADR(gc_DbmTranslation_de_Text2225), ADR(gc_DbmTranslation_de_Text2226), ADR(gc_DbmTranslation_de_Text2227), ADR(gc_DbmTranslation_de_Text2228), ADR(gc_DbmTranslation_de_Text2229), ADR(gc_DbmTranslation_de_Text2230), ADR(gc_DbmTranslation_de_Text2231), ADR(gc_DbmTranslation_de_Text2232), ADR(gc_DbmTranslation_de_Text2233), ADR(gc_DbmTranslation_de_Text2234), ADR(gc_DbmTranslation_de_Text2235), ADR(gc_DbmTranslation_de_Text2236), ADR(gc_DbmTranslation_de_Text2237), ADR(gc_DbmTranslation_de_Text2238), ADR(gc_DbmTranslation_de_Text2239), ADR(gc_DbmTranslation_de_Text2240), ADR(gc_DbmTranslation_de_Text2241), ADR(gc_DbmTranslation_de_Text2242), ADR(gc_DbmTranslation_de_Text2243), ADR(gc_DbmTranslation_de_Text2244), ADR(gc_DbmTranslation_de_Text2245), ADR(gc_DbmTranslation_de_Text2246), ADR(gc_DbmTranslation_de_Text2247), ADR(gc_DbmTranslation_de_Text2248), ADR(gc_DbmTranslation_de_Text2249), ADR(gc_DbmTranslation_de_Text2250), ADR(gc_DbmTranslation_de_Text2251), ADR(gc_DbmTranslation_de_Text2252), ADR(gc_DbmTranslation_de_Text2253), ADR(gc_DbmTranslation_de_Text2254), ADR(gc_DbmTranslation_de_Text2255), ADR(gc_DbmTranslation_de_Text2256), ADR(gc_DbmTranslation_de_Text2257), ADR(gc_DbmTranslation_de_Text2258), ADR(gc_DbmTranslation_de_Text2259), ADR(gc_DbmTranslation_de_Text2260), ADR(gc_DbmTranslation_de_Text2261), ADR(gc_DbmTranslation_de_Text2262), ADR(gc_DbmTranslation_de_Text2263), ADR(gc_DbmTranslation_de_Text2264), ADR(gc_DbmTranslation_de_Text2265), ADR(gc_DbmTranslation_de_Text2266), ADR(gc_DbmTranslation_de_Text2267), ADR(gc_DbmTranslation_de_Text2268), ADR(gc_DbmTranslation_de_Text2269), ADR(gc_DbmTranslation_de_Text2270), ADR(gc_DbmTranslation_de_Text2271), ADR(gc_DbmTranslation_de_Text2272), ADR(gc_DbmTranslation_de_Text2273), ADR(gc_DbmTranslation_de_Text2274), ADR(gc_DbmTranslation_de_Text2275), ADR(gc_DbmTranslation_de_Text2276), ADR(gc_DbmTranslation_de_Text2277), ADR(gc_DbmTranslation_de_Text2278), ADR(gc_DbmTranslation_de_Text2279), ADR(gc_DbmTranslation_de_Text2280), ADR(gc_DbmTranslation_de_Text2281), ADR(gc_DbmTranslation_de_Text2282), ADR(gc_DbmTranslation_de_Text2283), ADR(gc_DbmTranslation_de_Text2284), ADR(gc_DbmTranslation_de_Text2285), ADR(gc_DbmTranslation_de_Text2286), ADR(gc_DbmTranslation_de_Text2287), ADR(gc_DbmTranslation_de_Text2288), ADR(gc_DbmTranslation_de_Text2289), ADR(gc_DbmTranslation_de_Text2290), ADR(gc_DbmTranslation_de_Text2291), ADR(gc_DbmTranslation_de_Text2292), ADR(gc_DbmTranslation_de_Text2293), ADR(gc_DbmTranslation_de_Text2294), ADR(gc_DbmTranslation_de_Text2295), ADR(gc_DbmTranslation_de_Text2296), ADR(gc_DbmTranslation_de_Text2297), ADR(gc_DbmTranslation_de_Text2298), ADR(gc_DbmTranslation_de_Text2299), ADR(gc_DbmTranslation_de_Text2300), ADR(gc_DbmTranslation_de_Text2301), ADR(gc_DbmTranslation_de_Text2302), ADR(gc_DbmTranslation_de_Text2303), ADR(gc_DbmTranslation_de_Text2304), ADR(gc_DbmTranslation_de_Text2305), ADR(gc_DbmTranslation_de_Text2306), ADR(gc_DbmTranslation_de_Text2307), ADR(gc_DbmTranslation_de_Text2308), ADR(gc_DbmTranslation_de_Text2309), ADR(gc_DbmTranslation_de_Text2310), ADR(gc_DbmTranslation_de_Text2311), ADR(gc_DbmTranslation_de_Text2312), ADR(gc_DbmTranslation_de_Text2313), ADR(gc_DbmTranslation_de_Text2314), ADR(gc_DbmTranslation_de_Text2315), ADR(gc_DbmTranslation_de_Text2316), ADR(gc_DbmTranslation_de_Text2317), ADR(gc_DbmTranslation_de_Text2318), ADR(gc_DbmTranslation_de_Text2319), ADR(gc_DbmTranslation_de_Text2320), ADR(gc_DbmTranslation_de_Text2321), ADR(gc_DbmTranslation_de_Text2322), ADR(gc_DbmTranslation_de_Text2323), ADR(gc_DbmTranslation_de_Text2324), ADR(gc_DbmTranslation_de_Text2325), ADR(gc_DbmTranslation_de_Text2326), ADR(gc_DbmTranslation_de_Text2327), ADR(gc_DbmTranslation_de_Text2328), ADR(gc_DbmTranslation_de_Text2329), ADR(gc_DbmTranslation_de_Text2330), ADR(gc_DbmTranslation_de_Text2331), ADR(gc_DbmTranslation_de_Text2332), ADR(gc_DbmTranslation_de_Text2333), ADR(gc_DbmTranslation_de_Text2334), ADR(gc_DbmTranslation_de_Text2335), ADR(gc_DbmTranslation_de_Text2336), ADR(gc_DbmTranslation_de_Text2337), ADR(gc_DbmTranslation_de_Text2338), ADR(gc_DbmTranslation_de_Text2339), ADR(gc_DbmTranslation_de_Text2340), ADR(gc_DbmTranslation_de_Text2341), ADR(gc_DbmTranslation_de_Text2342), ADR(gc_DbmTranslation_de_Text2343), ADR(gc_DbmTranslation_de_Text2344), ADR(gc_DbmTranslation_de_Text2345), ADR(gc_DbmTranslation_de_Text2346), ADR(gc_DbmTranslation_de_Text2347), ADR(gc_DbmTranslation_de_Text2348), ADR(gc_DbmTranslation_de_Text2349), ADR(gc_DbmTranslation_de_Text2350), ADR(gc_DbmTranslation_de_Text2351), ADR(gc_DbmTranslation_de_Text2352), ADR(gc_DbmTranslation_de_Text2353), ADR(gc_DbmTranslation_de_Text2354), ADR(gc_DbVarGrpNameTranslation_de_Text2355), ADR(gc_DbVarGrpNameTranslation_de_Text2356), ADR(gc_DbVarGrpNameTranslation_de_Text2357), ADR(gc_DbVarGrpNameTranslation_de_Text2358), ADR(gc_DbVarGrpNameTranslation_de_Text2359), ADR(gc_DbVarGrpNameTranslation_de_Text2360), ADR(gc_DbVarGrpNameTranslation_de_Text2361), ADR(gc_DbVarGrpNameTranslation_de_Text2362), ADR(gc_DbVarGrpNameTranslation_de_Text2363), ADR(gc_DbVarGrpNameTranslation_de_Text2364), ADR(gc_DbVarGrpNameTranslation_de_Text2365), ADR(gc_DbVarGrpNameTranslation_de_Text2366), ADR(gc_DbVarGrpNameTranslation_de_Text2367), ADR(gc_DbVarGrpNameTranslation_de_Text2368), ADR(gc_DbVarGrpNameTranslation_de_Text2369), ADR(gc_DbVarGrpNameTranslation_de_Text2370), ADR(gc_DbVarGrpNameTranslation_de_Text2371)];
  gc_DbmTranslation_de : TTranslation := (IsoCode := 'de', EnglishName := "german", NativeName := "german", Texts := ADR(gc_DbmTranslation_de_Texts));
  gc_DbmTranslation_en_Text0 : WSTRING(39) := "Pressure Block Oscillation Sensor State";
  gc_DbmTranslation_en_Text1 : WSTRING(39) := "Pressure Block Oscillation Sensor Value";
  gc_DbmTranslation_en_Text2 : WSTRING(43) := "Pressure Block Oscillation Sensor Raw value";
  gc_DbmTranslation_en_Text3 : WSTRING(27) := "Pressure Brake Sensor State";
  gc_DbmTranslation_en_Text4 : WSTRING(27) := "Pressure Brake Sensor Value";
  gc_DbmTranslation_en_Text5 : WSTRING(31) := "Pressure Brake Sensor Raw value";
  gc_DbmTranslation_en_Text6 : WSTRING(37) := "Temperature Transmission Sensor State";
  gc_DbmTranslation_en_Text7 : WSTRING(37) := "Temperature Transmission Sensor Value";
  gc_DbmTranslation_en_Text8 : WSTRING(41) := "Temperature Transmission Sensor Raw value";
  gc_DbmTranslation_en_Text9 : WSTRING(25) := "Fault Pvg Left Trak State";
  gc_DbmTranslation_en_Text10 : WSTRING(29) := "Fault Pvg Left Trak Raw Value";
  gc_DbmTranslation_en_Text11 : WSTRING(26) := "Fault Pvg Right Trak State";
  gc_DbmTranslation_en_Text12 : WSTRING(30) := "Fault Pvg Right Trak Raw value";
  gc_DbmTranslation_en_Text13 : WSTRING(25) := "Down Axle oscillant State";
  gc_DbmTranslation_en_Text14 : WSTRING(39) := "Down Axle oscillant  Raw value pin 0 Nc";
  gc_DbmTranslation_en_Text15 : WSTRING(39) := "Down Axle oscillant  Raw value pin 1 No";
  gc_DbmTranslation_en_Text16 : WSTRING(20) := "Down Axle fixe state";
  gc_DbmTranslation_en_Text17 : WSTRING(24) := "Down Axle fixe Raw value";
  gc_DbmTranslation_en_Text18 : WSTRING(33) := "Down Axle fixe Raw value pin 1 No";
  gc_DbmTranslation_en_Text19 : WSTRING(23) := "Up Axle oscillant state";
  gc_DbmTranslation_en_Text20 : WSTRING(23) := "Up Axle oscillant value";
  gc_DbmTranslation_en_Text21 : WSTRING(18) := "Up Axle fixe state";
  gc_DbmTranslation_en_Text22 : WSTRING(22) := "Up Axle fixe raw value";
  gc_DbmTranslation_en_Text23 : WSTRING(29) := "Frame rotation sensor 1 state";
  gc_DbmTranslation_en_Text24 : WSTRING(33) := "Frame rotation sensor 1 raw value";
  gc_DbmTranslation_en_Text25 : WSTRING(39) := "Frame rotation sensor 1 raw value Pin 1";
  gc_DbmTranslation_en_Text26 : WSTRING(22) := "Rail hook sensor state";
  gc_DbmTranslation_en_Text27 : WSTRING(26) := "Rail hook sensor raw value";
  gc_DbmTranslation_en_Text28 : WSTRING(27) := "Inductive Rail sensor state";
  gc_DbmTranslation_en_Text29 : WSTRING(31) := "Inductive Rail sensor raw value";
  gc_DbmTranslation_en_Text30 : WSTRING(21) := "Centered turret state";
  gc_DbmTranslation_en_Text31 : WSTRING(25) := "Centered turret raw value";
  gc_DbmTranslation_en_Text32 : WSTRING(25) := "Work Key track Side state";
  gc_DbmTranslation_en_Text33 : WSTRING(29) := "Work Key track Side raw value";
  gc_DbmTranslation_en_Text34 : WSTRING(29) := "Frame rotation sensor 2 state";
  gc_DbmTranslation_en_Text35 : WSTRING(39) := "Frame rotation sensor 2 raw value Pin 0";
  gc_DbmTranslation_en_Text36 : WSTRING(39) := "Frame rotation sensor 2 raw value Pin 1";
  gc_DbmTranslation_en_Text37 : WSTRING(24) := "Work Key Bilateral state";
  gc_DbmTranslation_en_Text38 : WSTRING(28) := "Work Key Bilateral raw value";
  gc_DbmTranslation_en_Text39 : WSTRING(22) := "Work Key Centred state";
  gc_DbmTranslation_en_Text40 : WSTRING(26) := "Work Key Centred raw value";
  gc_DbmTranslation_en_Text41 : WSTRING(32) := "Abutment turret track side state";
  gc_DbmTranslation_en_Text42 : WSTRING(36) := "Abutment turret track side raw value";
  gc_DbmTranslation_en_Text43 : WSTRING(34) := "Abutment Turret Centred Side state";
  gc_DbmTranslation_en_Text44 : WSTRING(38) := "Abutment Turret Centred Side raw value";
  gc_DbmTranslation_en_Text45 : WSTRING(43) := "Oscillant Axle Speed Sensor Direction state";
  gc_DbmTranslation_en_Text46 : WSTRING(47) := "Oscillant Axle Speed Sensor Direction Raw value";
  gc_DbmTranslation_en_Text47 : WSTRING(38) := "Fixe Axle Speed Sensor Direction state";
  gc_DbmTranslation_en_Text48 : WSTRING(42) := "Fixe Axle Speed Sensor Direction Raw value";
  gc_DbmTranslation_en_Text49 : WSTRING(19) := "Trailer gache state";
  gc_DbmTranslation_en_Text50 : WSTRING(23) := "Trailer gache raw value";
  gc_DbmTranslation_en_Text51 : WSTRING(34) := "Measuring mast sensor folded state";
  gc_DbmTranslation_en_Text52 : WSTRING(38) := "Measuring mast sensor folded raw value";
  gc_DbmTranslation_en_Text53 : WSTRING(24) := "Oscillant Axle frequency";
  gc_DbmTranslation_en_Text54 : WSTRING(19) := "Fixe Axle frequency";
  gc_DbmTranslation_en_Text55 : WSTRING(25) := "Aru Radio 1 Contact state";
  gc_DbmTranslation_en_Text56 : WSTRING(29) := "Aru Radio 1 Contact raw value";
  gc_DbmTranslation_en_Text57 : WSTRING(25) := "Aru Radio 2 Contact state";
  gc_DbmTranslation_en_Text58 : WSTRING(29) := "Aru Radio 2 Contact raw value";
  gc_DbmTranslation_en_Text59 : WSTRING(19) := "Aru 1 Contact state";
  gc_DbmTranslation_en_Text60 : WSTRING(23) := "Aru 1 Contact raw value";
  gc_DbmTranslation_en_Text61 : WSTRING(19) := "Aru 2 Contact state";
  gc_DbmTranslation_en_Text62 : WSTRING(23) := "Aru 2 contact raw value";
  gc_DbmTranslation_en_Text63 : WSTRING(19) := "Starter motor state";
  gc_DbmTranslation_en_Text64 : WSTRING(23) := "Starter motor raw value";
  gc_DbmTranslation_en_Text65 : WSTRING(33) := "Autorisation High Speed Key State";
  gc_DbmTranslation_en_Text66 : WSTRING(37) := "Autorisation High Speed Key Raw Value";
  gc_DbmTranslation_en_Text67 : WSTRING(35) := "Electric pump Pressure Sensor State";
  gc_DbmTranslation_en_Text68 : WSTRING(35) := "Electric pump Pressure Sensor Value";
  gc_DbmTranslation_en_Text69 : WSTRING(39) := "Electric pump Pressure Sensor Raw value";
  gc_DbmTranslation_en_Text70 : WSTRING(29) := "Mast sensor position UP State";
  gc_DbmTranslation_en_Text71 : WSTRING(33) := "Mast sensor position UP Raw Value";
  gc_DbmTranslation_en_Text72 : WSTRING(46) := "Hydraulic valve uin down position sensor state";
  gc_DbmTranslation_en_Text73 : WSTRING(50) := "Hydraulic valve uin down position sensor raw value";
  gc_DbmTranslation_en_Text74 : WSTRING(33) := "Ev Deflector Transmission command";
  gc_DbmTranslation_en_Text75 : WSTRING(38) := "Ev Deflector Transmission actual value";
  gc_DbmTranslation_en_Text76 : WSTRING(28) := "Ev Up Measuring Mast command";
  gc_DbmTranslation_en_Text77 : WSTRING(33) := "Ev Up Measuring Mast actual value";
  gc_DbmTranslation_en_Text78 : WSTRING(30) := "Ev Down Measuring Mast command";
  gc_DbmTranslation_en_Text79 : WSTRING(35) := "Ev Down Measuring Mast actual value";
  gc_DbmTranslation_en_Text80 : WSTRING(30) := "Ev Service Brake Track command";
  gc_DbmTranslation_en_Text81 : WSTRING(35) := "Ev Service Brake Track actual value";
  gc_DbmTranslation_en_Text82 : WSTRING(26) := "Ev Power Reduction command";
  gc_DbmTranslation_en_Text83 : WSTRING(31) := "Ev Power Reduction actual value";
  gc_DbmTranslation_en_Text84 : WSTRING(27) := "Ev Frame Rotation 1 command";
  gc_DbmTranslation_en_Text85 : WSTRING(32) := "Ev Frame Rotation 1 actual value";
  gc_DbmTranslation_en_Text86 : WSTRING(27) := "Ev Frame Rotation 2 command";
  gc_DbmTranslation_en_Text87 : WSTRING(32) := "Ev Frame Rotation 2 actual value";
  gc_DbmTranslation_en_Text88 : WSTRING(29) := "Supply Radio Receiver command";
  gc_DbmTranslation_en_Text89 : WSTRING(34) := "Supply Radio Receiver actual value";
  gc_DbmTranslation_en_Text90 : WSTRING(34) := "Buzzer Lynx Moving Machine command";
  gc_DbmTranslation_en_Text91 : WSTRING(39) := "Buzzer Lynx Moving Machine actual value";
  gc_DbmTranslation_en_Text92 : WSTRING(28) := "White Lights Trailer command";
  gc_DbmTranslation_en_Text93 : WSTRING(33) := "White Lights Trailer actual value";
  gc_DbmTranslation_en_Text94 : WSTRING(26) := "Red Lights Trailer command";
  gc_DbmTranslation_en_Text95 : WSTRING(31) := "Red Lights Trailer actual value";
  gc_DbmTranslation_en_Text96 : WSTRING(23) := "White Light AVG command";
  gc_DbmTranslation_en_Text97 : WSTRING(28) := "White Light AVG actual value";
  gc_DbmTranslation_en_Text98 : WSTRING(23) := "White Light AVD command";
  gc_DbmTranslation_en_Text99 : WSTRING(28) := "White Light AVD actual value";
  gc_DbmTranslation_en_Text100 : WSTRING(21) := "Red Light AVG command";
  gc_DbmTranslation_en_Text101 : WSTRING(26) := "Red Light AVG actual value";
  gc_DbmTranslation_en_Text102 : WSTRING(21) := "Red Light AVD command";
  gc_DbmTranslation_en_Text103 : WSTRING(26) := "Red Light AVD actual value";
  gc_DbmTranslation_en_Text104 : WSTRING(23) := "White Light ARG command";
  gc_DbmTranslation_en_Text105 : WSTRING(28) := "White Light ARG actual value";
  gc_DbmTranslation_en_Text106 : WSTRING(23) := "White Light ARD command";
  gc_DbmTranslation_en_Text107 : WSTRING(28) := "White Light ARD actual value";
  gc_DbmTranslation_en_Text108 : WSTRING(21) := "Red Light ARG command";
  gc_DbmTranslation_en_Text109 : WSTRING(26) := "Red Light ARG actual value";
  gc_DbmTranslation_en_Text110 : WSTRING(21) := "Red Light ARD command";
  gc_DbmTranslation_en_Text111 : WSTRING(26) := "Red Light ARD actual value";
  gc_DbmTranslation_en_Text112 : WSTRING(29) := "Suplly Pvg Left Track command";
  gc_DbmTranslation_en_Text113 : WSTRING(34) := "Suplly Pvg Left Track actual value";
  gc_DbmTranslation_en_Text114 : WSTRING(30) := "Suplly Pvg Right Track command";
  gc_DbmTranslation_en_Text115 : WSTRING(35) := "Suplly Pvg Right Track actual value";
  gc_DbmTranslation_en_Text116 : WSTRING(33) := "Ev UnBlock Oscillation Axle state";
  gc_DbmTranslation_en_Text117 : WSTRING(40) := "Ev UnBlock Oscillation Axle command bool";
  gc_DbmTranslation_en_Text118 : WSTRING(26) := "Ev Up Axle Oscillant state";
  gc_DbmTranslation_en_Text119 : WSTRING(33) := "Ev Up Axle Oscillant Command Bool";
  gc_DbmTranslation_en_Text120 : WSTRING(29) := "Ev Down Axle Oscillant  state";
  gc_DbmTranslation_en_Text121 : WSTRING(35) := "Ev Down Axle Oscillant Command Bool";
  gc_DbmTranslation_en_Text122 : WSTRING(20) := "Ev Up AxleFixe state";
  gc_DbmTranslation_en_Text123 : WSTRING(28) := "Ev Up Axle Fixe Command Bool";
  gc_DbmTranslation_en_Text124 : WSTRING(22) := "Ev Down AxleFixe state";
  gc_DbmTranslation_en_Text125 : WSTRING(30) := "Ev Down Axle Fixe Command Bool";
  gc_DbmTranslation_en_Text126 : WSTRING(35) := "Ev Park Brake Axle Oscillant  state";
  gc_DbmTranslation_en_Text127 : WSTRING(42) := "Ev Park Brake Axle Oscillant  command bool";
  gc_DbmTranslation_en_Text128 : WSTRING(29) := "Ev Park Brake Axle Fixe state";
  gc_DbmTranslation_en_Text129 : WSTRING(37) := "Ev Park Brake Axle Fixe  command bool";
  gc_DbmTranslation_en_Text130 : WSTRING(37) := "Ev Service Brake Axle Oscillant state";
  gc_DbmTranslation_en_Text131 : WSTRING(36) := "Ev Service Brake Axle 1 command Bool";
  gc_DbmTranslation_en_Text132 : WSTRING(32) := "Ev Service Brake Axle Fixe state";
  gc_DbmTranslation_en_Text133 : WSTRING(36) := "Ev Service Brake Axle 2 command Bool";
  gc_DbmTranslation_en_Text134 : WSTRING(19) := "Klaxon Neotec state";
  gc_DbmTranslation_en_Text135 : WSTRING(26) := "Klaxon Neotec command bool";
  gc_DbmTranslation_en_Text136 : WSTRING(18) := "Forward pump state";
  gc_DbmTranslation_en_Text137 : WSTRING(21) := "Forward pump  command";
  gc_DbmTranslation_en_Text138 : WSTRING(27) := "Forward pump actual current";
  gc_DbmTranslation_en_Text139 : WSTRING(19) := "Backward pump state";
  gc_DbmTranslation_en_Text140 : WSTRING(22) := "Backward pump  command";
  gc_DbmTranslation_en_Text141 : WSTRING(28) := "Backward pump actual current";
  gc_DbmTranslation_en_Text142 : WSTRING(22) := "Pvg left track command";
  gc_DbmTranslation_en_Text143 : WSTRING(29) := "Pvg left track actual voltage";
  gc_DbmTranslation_en_Text144 : WSTRING(23) := "Pvg right track command";
  gc_DbmTranslation_en_Text145 : WSTRING(30) := "Pvg right track actual voltage";
  gc_DbmTranslation_en_Text146 : WSTRING(26) := "Supply Ana Sensors Command";
  gc_DbmTranslation_en_Text147 : WSTRING(24) := "Supply Ana Sensors Value";
  gc_DbmTranslation_en_Text148 : WSTRING(30) := "Pvg Left Track Lowside Command";
  gc_DbmTranslation_en_Text149 : WSTRING(28) := "Pvg Left Track Lowside Value";
  gc_DbmTranslation_en_Text150 : WSTRING(31) := "Pvg Right Track Lowside Command";
  gc_DbmTranslation_en_Text151 : WSTRING(29) := "Pvg Right Track Lowside Value";
  gc_DbmTranslation_en_Text152 : WSTRING(39) := "Return low side Ev Forward Pump command";
  gc_DbmTranslation_en_Text153 : WSTRING(37) := "Return low side Ev Forward Pump state";
  gc_DbmTranslation_en_Text154 : WSTRING(40) := "Return low side Ev Backward Pump command";
  gc_DbmTranslation_en_Text155 : WSTRING(38) := "Return low side Ev Backward Pump state";
  gc_DbmTranslation_en_Text156 : WSTRING(19) := "Neon Lights command";
  gc_DbmTranslation_en_Text157 : WSTRING(17) := "Neon Lights value";
  gc_DbmTranslation_en_Text158 : WSTRING(33) := "Ev 2 Deflector Transmission value";
  gc_DbmTranslation_en_Text159 : WSTRING(21) := "Cooling relay command";
  gc_DbmTranslation_en_Text160 : WSTRING(19) := "Cooling relay state";
  gc_DbmTranslation_en_Text161 : WSTRING(54) := "Sorties d’activation de l’Ev du deuxième frein de parc";
  gc_DbmTranslation_en_Text162 : WSTRING(54) := "Sorties d’activation de l’Ev du deuxième frein de parc";
  gc_DbmTranslation_en_Text163 : WSTRING(33) := "Ev 2nd Park Brake Axle Fixe State";
  gc_DbmTranslation_en_Text164 : WSTRING(33) := "Ev 2nd Park Brake Axle Osci State";
  gc_DbmTranslation_en_Text165 : WSTRING(41) := "Pvg Translation for Rail Electric Command";
  gc_DbmTranslation_en_Text166 : WSTRING(41) := "Pvg Translation for Rail Electric Voltage";
  gc_DbmTranslation_en_Text167 : WSTRING(48) := "Suplly Pvg Translation for Rail Electric Command";
  gc_DbmTranslation_en_Text168 : WSTRING(46) := "Suplly Pvg Translation for Rail Electric State";
  gc_DbmTranslation_en_Text169 : WSTRING(42) := "Ev Deviator for Rail Electric Mode Command";
  gc_DbmTranslation_en_Text170 : WSTRING(40) := "Ev Deviator for Rail Electric Mode State";
  gc_DbmTranslation_en_Text171 : WSTRING(43) := "Relay Cut Off Variator for Electric Command";
  gc_DbmTranslation_en_Text172 : WSTRING(41) := "Relay Cut Off Variator for Electric State";
  gc_DbmTranslation_en_Text173 : WSTRING(28) := "Relay Enable Battery Command";
  gc_DbmTranslation_en_Text174 : WSTRING(26) := "Relay Enable Battery State";
  gc_DbmTranslation_en_Text175 : WSTRING(25) := "Byte increased each cycle";
  gc_DbmTranslation_en_Text176 : WSTRING(22) := "Watchdog current state";
  gc_DbmTranslation_en_Text177 : WSTRING(11) := "Ecu voltage";
  gc_DbmTranslation_en_Text178 : WSTRING(13) := "Off Rail Mode";
  gc_DbmTranslation_en_Text179 : WSTRING(9) := "Rail Mode";
  gc_DbmTranslation_en_Text180 : WSTRING(75) := "Output value Lut of Manipulator left radio control in range -10000 to 10000";
  gc_DbmTranslation_en_Text181 : WSTRING(35) := "Output value Lut of Left Track Pvg ";
  gc_DbmTranslation_en_Text182 : WSTRING(76) := "Output value Lut of Manipulator Right radio control in range -10000 to 10000";
  gc_DbmTranslation_en_Text183 : WSTRING(36) := "Output value Lut of Right Track Pvg ";
  gc_DbmTranslation_en_Text184 : WSTRING(52) := "Outût value Lut of Joystick advance Rail translation";
  gc_DbmTranslation_en_Text185 : WSTRING(40) := "Output Lut  of Forward Pump Transmission";
